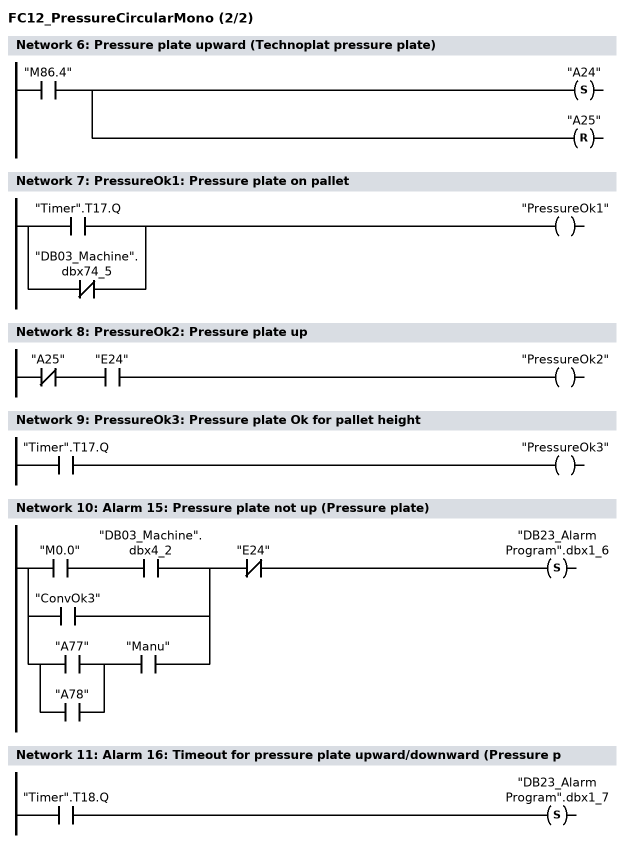
   RUNG wire#powerrail
      Contact( "M86.4" )
      wire#w1
      S_Coil( "A24" )
   END_RUNG
   RUNG wire#w1
      R_Coil( "A25" )
   END_RUNG
   // the same network as SCL:
   IF "M86.4" THEN
       "A24" := TRUE;
       "A25" := FALSE;
   END_IF;
END_REGION

REGION Network 7: PressureOk1: Pressure plate on pallet
   RUNG wire#powerrail
      Contact( "Timer".T17.Q )
      wire#w1
      Coil( "PressureOk1" )
   END_RUNG
   RUNG wire#powerrail
      I_Contact( "DB03_Machine".dbx74_5 )
   END_RUNG wire#w1
   // the same network as SCL:
   "PressureOk1" := "Timer".T17.Q OR NOT "DB03_Machine".dbx74_5;
END_REGION

REGION Network 8: PressureOk2: Pressure plate up
   RUNG wire#powerrail
      I_Contact( "A25" )
      Contact( "E24" )
      Coil( "PressureOk2" )
   END_RUNG
   // the same network as SCL:
   "PressureOk2" := NOT "A25" AND "E24";
END_REGION

REGION Network 9: PressureOk3: Pressure plate Ok for pallet height
   RUNG wire#powerrail
      Contact( "Timer".T17.Q )
      Coil( "PressureOk3" )
   END_RUNG
   // the same network as SCL:
   "PressureOk3" := "Timer".T17.Q;
END_REGION

REGION Network 10: Alarm 15: Pressure plate not up (Pressure plate)
   RUNG wire#powerrail
      Contact( "M0.0" )
      Contact( "DB03_Machine".dbx4_2 )
      wire#w1
      I_Contact( "E24" )
      S_Coil( "DB23_AlarmProgram".dbx1_6 )
   END_RUNG
   RUNG wire#powerrail
      Contact( "ConvOk3" )
   END_RUNG wire#w1
   RUNG wire#powerrail
      Contact( "A77" )
      wire#w2
      Contact( "Manu" )
   END_RUNG wire#w1
   RUNG wire#powerrail
      Contact( "A78" )
   END_RUNG wire#w2
   // the same network as SCL:
   IF (("M0.0" AND "DB03_Machine".dbx4_2) OR "ConvOk3" OR (("A77" OR "A78") AND "Manu")) AND NOT "E24" THEN
       "DB23_AlarmProgram".dbx1_6 := TRUE;
   END_IF;
END_REGION

REGION Network 11: Alarm 16: Timeout for pressure plate upward/downward (Pressure p
   RUNG wire#powerrail
      Contact( "Timer".T18.Q )
      S_Coil( "DB23_AlarmProgram".dbx1_7 )
   END_RUNG
   // the same network as SCL:
   IF "Timer".T18.Q THEN "DB23_AlarmProgram".dbx1_7 := TRUE; END_IF;
END_REGION
END_FUNCTION

FUNCTION "FC26_Pos1SensorDec" : Void   // FC26, LAD
{ S7_Optimized_Access := 'FALSE' }
VERSION : 0.1
// stored: AutoNumber false, IsIECCheckEnabled false, SetENOAutomatically false, UDAEnableTagReadback false
BEGIN

REGION Network 1: Delay on pallet positioning
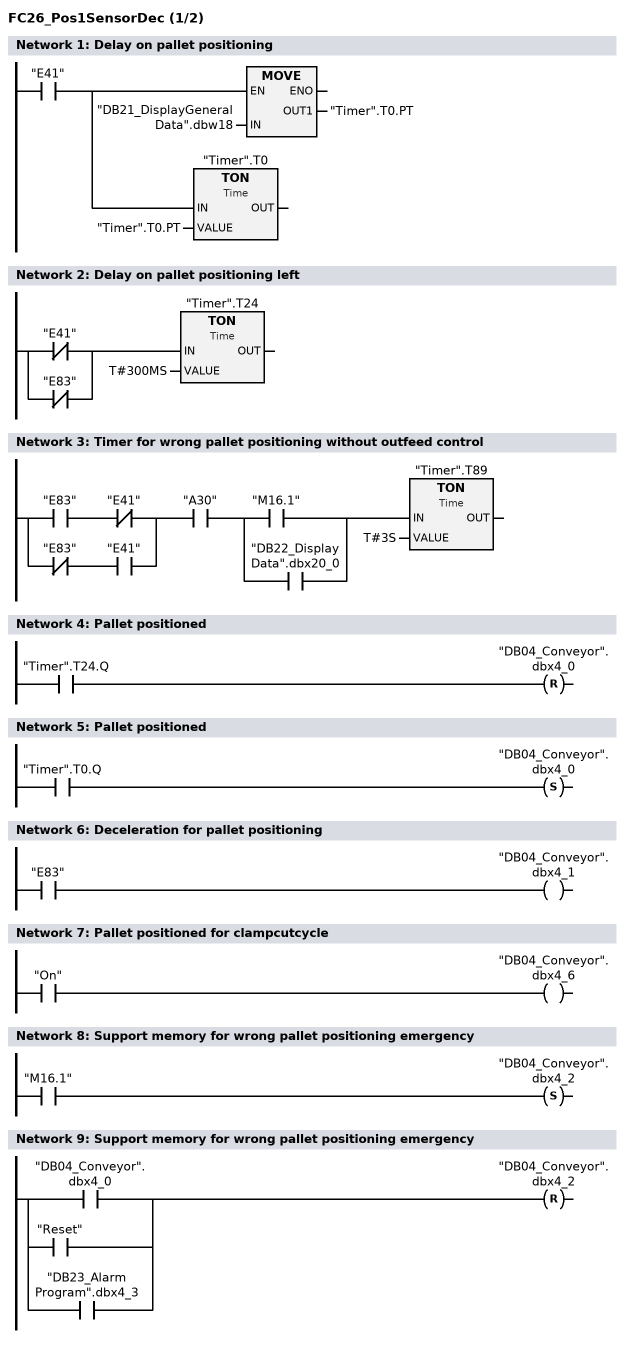
   IF "E41" THEN "Timer".T0.PT := "DB21_DisplayGeneralData".dbw18; END_IF;
   "Timer".T0.TON(IN := "E41", PT := "Timer".T0.PT);   // TON coil
END_REGION

REGION Network 2: Delay on pallet positioning left
   "Timer".T24.TON(IN := NOT "E41" OR NOT "E83", PT := T#300MS);   // TON coil
END_REGION

REGION Network 3: Timer for wrong pallet positioning without outfeed control
   "Timer".T89.TON(IN := (("E83" AND NOT "E41") OR (NOT "E83" AND "E41")) AND "A30" AND ("M16.1" OR "DB22_DisplayData".dbx20_0), PT := T#3S);   // TON coil
END_REGION

REGION Network 4: Pallet positioned
   RUNG wire#powerrail
      Contact( "Timer".T24.Q )
      R_Coil( "DB04_Conveyor".dbx4_0 )
   END_RUNG
   // the same network as SCL:
   IF "Timer".T24.Q THEN "DB04_Conveyor".dbx4_0 := FALSE; END_IF;
END_REGION

REGION Network 5: Pallet positioned
   RUNG wire#powerrail
      Contact( "Timer".T0.Q )
      S_Coil( "DB04_Conveyor".dbx4_0 )
   END_RUNG
   // the same network as SCL:
   IF "Timer".T0.Q THEN "DB04_Conveyor".dbx4_0 := TRUE; END_IF;
END_REGION

REGION Network 6: Deceleration for pallet positioning
   RUNG wire#powerrail
      Contact( "E83" )
      Coil( "DB04_Conveyor".dbx4_1 )
   END_RUNG
   // the same network as SCL:
   "DB04_Conveyor".dbx4_1 := "E83";
END_REGION

REGION Network 7: Pallet positioned for clampcutcycle
   RUNG wire#powerrail
      Contact( "On" )
      Coil( "DB04_Conveyor".dbx4_6 )
   END_RUNG
   // the same network as SCL:
   "DB04_Conveyor".dbx4_6 := "On";
END_REGION

REGION Network 8: Support memory for wrong pallet positioning emergency
   RUNG wire#powerrail
      Contact( "M16.1" )
      S_Coil( "DB04_Conveyor".dbx4_2 )
   END_RUNG
   // the same network as SCL:
   IF "M16.1" THEN "DB04_Conveyor".dbx4_2 := TRUE; END_IF;
END_REGION

REGION Network 9: Support memory for wrong pallet positioning emergency
   RUNG wire#powerrail
      Contact( "DB04_Conveyor".dbx4_0 )
      wire#w1
      R_Coil( "DB04_Conveyor".dbx4_2 )
   END_RUNG
   RUNG wire#powerrail
      Contact( "Reset" )
   END_RUNG wire#w1
   RUNG wire#powerrail
      Contact( "DB23_AlarmProgram".dbx4_3 )
   END_RUNG wire#w1
   // the same network as SCL:
   IF "DB04_Conveyor".dbx4_0 OR "Reset" OR "DB23_AlarmProgram".dbx4_3 THEN
       "DB04_Conveyor".dbx4_2 := FALSE;
   END_IF;
END_REGION

REGION Network 10: Alarm 33: Pallet positioning released during table rotation (Con
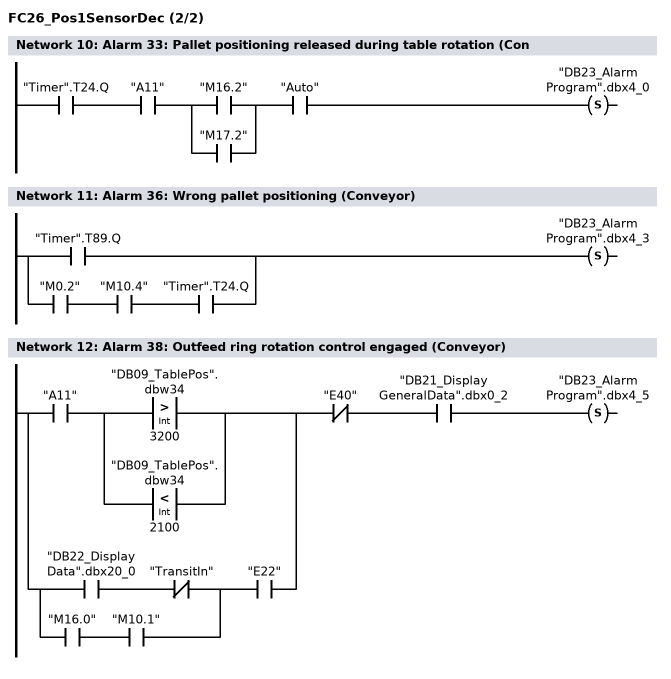
   RUNG wire#powerrail
      Contact( "Timer".T24.Q )
      Contact( "A11" )
      wire#w1
      Contact( "M16.2" )
      wire#w2
      Contact( "Auto" )
      S_Coil( "DB23_AlarmProgram".dbx4_0 )
   END_RUNG
   RUNG wire#w1
      Contact( "M17.2" )
   END_RUNG wire#w2
   // the same network as SCL:
   IF "Timer".T24.Q AND "A11" AND ("M16.2" OR "M17.2") AND "Auto" THEN
       "DB23_AlarmProgram".dbx4_0 := TRUE;
   END_IF;
END_REGION

REGION Network 11: Alarm 36: Wrong pallet positioning (Conveyor)
   RUNG wire#powerrail
      Contact( "Timer".T89.Q )
      wire#w1
      S_Coil( "DB23_AlarmProgram".dbx4_3 )
   END_RUNG
   RUNG wire#powerrail
      Contact( "M0.2" )
      Contact( "M10.4" )
      Contact( "Timer".T24.Q )
   END_RUNG wire#w1
   // the same network as SCL:
   IF "Timer".T89.Q OR ("M0.2" AND "M10.4" AND "Timer".T24.Q) THEN
       "DB23_AlarmProgram".dbx4_3 := TRUE;
   END_IF;
END_REGION

REGION Network 12: Alarm 38: Outfeed ring rotation control engaged (Conveyor)
   RUNG wire#powerrail
      Contact( "A11" )
      wire#w1
      { S7_Templates := "SrcType := Int" } GT_Contact(in1 := "DB09_TablePos".dbw34, in2 := 3200)
      wire#w2
      I_Contact( "E40" )
      Contact( "DB21_DisplayGeneralData".dbx0_2 )
      S_Coil( "DB23_AlarmProgram".dbx4_5 )
   END_RUNG
   RUNG wire#w1
      { S7_Templates := "SrcType := Int" } LT_Contact(in1 := "DB09_TablePos".dbw34, in2 := 2100)
   END_RUNG wire#w2
   RUNG wire#powerrail
      Contact( "DB22_DisplayData".dbx20_0 )
      I_Contact( "TransitIn" )
      wire#w3
      Contact( "E22" )
   END_RUNG wire#w2
   RUNG wire#powerrail
      Contact( "M16.0" )
      Contact( "M10.1" )
   END_RUNG wire#w3
   // the same network as SCL:
   IF (("A11" AND (("DB09_TablePos".dbw34 > 3200) OR ("DB09_TablePos".dbw34 < 2100))) OR ((("DB22_DisplayData".dbx20_0 AND NOT "TransitIn") OR ("M16.0" AND "M10.1")) AND "E22")) AND NOT "E40" AND "DB21_DisplayGeneralData".dbx0_2 THEN
       "DB23_AlarmProgram".dbx4_5 := TRUE;
   END_IF;
END_REGION
END_FUNCTION

FUNCTION "FC27_PosSelfcEncoder" : Void   // FC27, LAD
TITLE = Pallet positioning with selfcentering system and encoder
{ S7_Optimized_Access := 'FALSE' }
AUTHOR : Robopac
VERSION : 0.0
// stored: AutoNumber false, IsIECCheckEnabled false, SetENOAutomatically false, UDAEnableTagReadback false
   VAR_TEMP
      Ch7ValmmEnco1 : DInt;
      Ch7ValmmEnco2 : DInt;
      PalletLenghtdiv2 : Int;
      PosToReach : Int;
      PosToDecelation : Int;
      WTemp1 : Int;
      DWTemp1 : DInt;
      DWTemp2 : DInt;
   END_VAR
   VAR_TEMP   // added for the SCL form of the ladder/FBD networks
      _w1 : Bool;
      _w2 : Bool;
   END_VAR
BEGIN

REGION Network 1: Delay on pallet positioning left
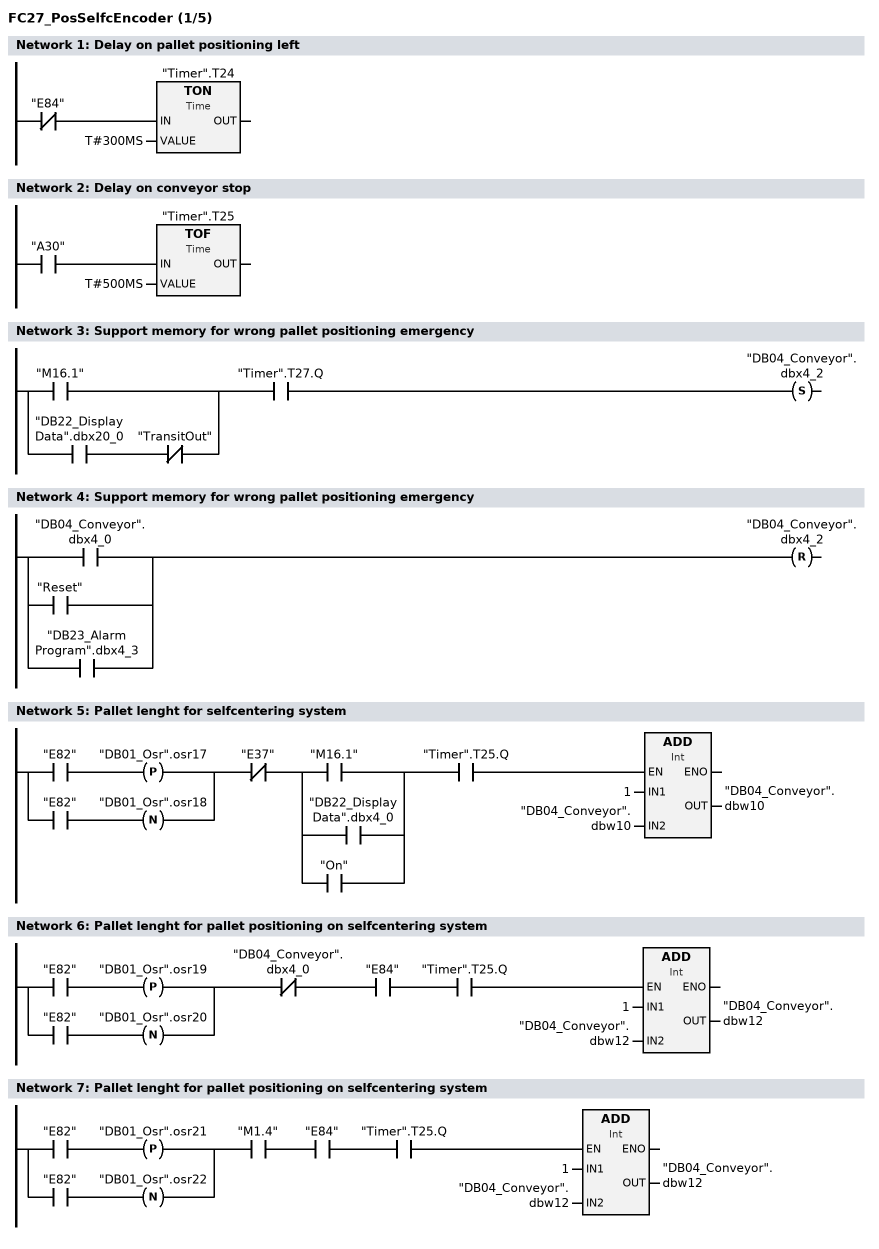
   "Timer".T24.TON(IN := NOT "E84", PT := T#300MS);   // TON coil
END_REGION

REGION Network 2: Delay on conveyor stop
   "Timer".T25.TOF(IN := "A30", PT := T#500MS);   // TOF coil
END_REGION

REGION Network 3: Support memory for wrong pallet positioning emergency
   RUNG wire#powerrail
      Contact( "M16.1" )
      wire#w1
      Contact( "Timer".T27.Q )
      S_Coil( "DB04_Conveyor".dbx4_2 )
   END_RUNG
   RUNG wire#powerrail
      Contact( "DB22_DisplayData".dbx20_0 )
      I_Contact( "TransitOut" )
   END_RUNG wire#w1
   // the same network as SCL:
   IF ("M16.1" OR ("DB22_DisplayData".dbx20_0 AND NOT "TransitOut")) AND "Timer".T27.Q THEN
       "DB04_Conveyor".dbx4_2 := TRUE;
   END_IF;
END_REGION

REGION Network 4: Support memory for wrong pallet positioning emergency
   RUNG wire#powerrail
      Contact( "DB04_Conveyor".dbx4_0 )
      wire#w1
      R_Coil( "DB04_Conveyor".dbx4_2 )
   END_RUNG
   RUNG wire#powerrail
      Contact( "Reset" )
   END_RUNG wire#w1
   RUNG wire#powerrail
      Contact( "DB23_AlarmProgram".dbx4_3 )
   END_RUNG wire#w1
   // the same network as SCL:
   IF "DB04_Conveyor".dbx4_0 OR "Reset" OR "DB23_AlarmProgram".dbx4_3 THEN
       "DB04_Conveyor".dbx4_2 := FALSE;
   END_IF;
END_REGION

REGION Network 5: Pallet lenght for selfcentering system
   RUNG wire#powerrail
      Contact( "E82" )
      P_Trig( "DB01_Osr".osr17 )
      wire#w1
      I_Contact( "E37" )
      wire#w2
      Contact( "M16.1" )
      wire#w3
      Contact( "Timer".T25.Q )
      { S7_Templates := "SrcType := Int"; S7_GenerateENO := "TRUE" } Add(in1 := 1, in2 := "DB04_Conveyor".dbw10, out => "DB04_Conveyor".dbw10)
   END_RUNG
   RUNG wire#powerrail
      Contact( "E82" )
      N_Trig( "DB01_Osr".osr18 )
   END_RUNG wire#w1
   RUNG wire#w2
      Contact( "DB22_DisplayData".dbx4_0 )
   END_RUNG wire#w3
   RUNG wire#w2
      Contact( "On" )
   END_RUNG wire#w3
   // the same network as SCL:
   #_w1 := "E82" AND NOT "DB01_Osr".osr17;   // rising edge
   "DB01_Osr".osr17 := "E82";
   #_w2 := NOT "E82" AND "DB01_Osr".osr18;   // falling edge
   "DB01_Osr".osr18 := "E82";
   IF (#_w1 OR #_w2) AND NOT "E37" AND ("M16.1" OR "DB22_DisplayData".dbx4_0 OR "On") AND "Timer".T25.Q THEN
       "DB04_Conveyor".dbw10 := 1 + "DB04_Conveyor".dbw10;
   END_IF;
END_REGION

REGION Network 6: Pallet lenght for pallet positioning on selfcentering system
   RUNG wire#powerrail
      Contact( "E82" )
      P_Trig( "DB01_Osr".osr19 )
      wire#w1
      I_Contact( "DB04_Conveyor".dbx4_0 )
      Contact( "E84" )
      Contact( "Timer".T25.Q )
      { S7_Templates := "SrcType := Int"; S7_GenerateENO := "TRUE" } Add(in1 := 1, in2 := "DB04_Conveyor".dbw12, out => "DB04_Conveyor".dbw12)
   END_RUNG
   RUNG wire#powerrail
      Contact( "E82" )
      N_Trig( "DB01_Osr".osr20 )
   END_RUNG wire#w1
   // the same network as SCL:
   #_w1 := "E82" AND NOT "DB01_Osr".osr19;   // rising edge
   "DB01_Osr".osr19 := "E82";
   #_w2 := NOT "E82" AND "DB01_Osr".osr20;   // falling edge
   "DB01_Osr".osr20 := "E82";
   IF (#_w1 OR #_w2) AND NOT "DB04_Conveyor".dbx4_0 AND "E84" AND "Timer".T25.Q THEN
       "DB04_Conveyor".dbw12 := 1 + "DB04_Conveyor".dbw12;
   END_IF;
END_REGION

REGION Network 7: Pallet lenght for pallet positioning on selfcentering system
   RUNG wire#powerrail
      Contact( "E82" )
      P_Trig( "DB01_Osr".osr21 )
      wire#w1
      Contact( "M1.4" )
      Contact( "E84" )
      Contact( "Timer".T25.Q )
      { S7_Templates := "SrcType := Int"; S7_GenerateENO := "TRUE" } Add(in1 := 1, in2 := "DB04_Conveyor".dbw12, out => "DB04_Conveyor".dbw12)
   END_RUNG
   RUNG wire#powerrail
      Contact( "E82" )
      N_Trig( "DB01_Osr".osr22 )
   END_RUNG wire#w1
   // the same network as SCL:
   #_w1 := "E82" AND NOT "DB01_Osr".osr21;   // rising edge
   "DB01_Osr".osr21 := "E82";
   #_w2 := NOT "E82" AND "DB01_Osr".osr22;   // falling edge
   "DB01_Osr".osr22 := "E82";
   IF (#_w1 OR #_w2) AND "M1.4" AND "E84" AND "Timer".T25.Q THEN
       "DB04_Conveyor".dbw12 := 1 + "DB04_Conveyor".dbw12;
   END_IF;
END_REGION

REGION Network 8: Reset pallet lenght
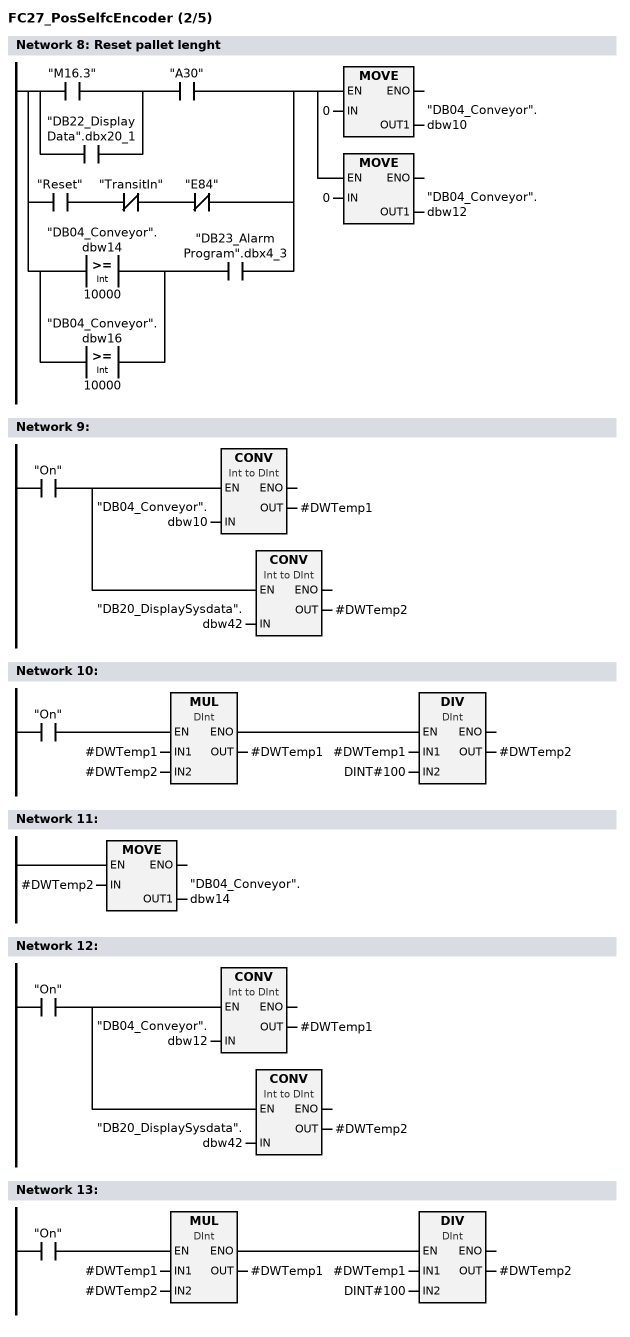
   RUNG wire#powerrail
      Contact( "M16.3" )
      wire#w1
      Contact( "A30" )
      wire#w2
      { S7_GenerateENO := "TRUE" } Move(in := 0, out1 => "DB04_Conveyor".dbw10)
   END_RUNG
   RUNG wire#powerrail
      Contact( "DB22_DisplayData".dbx20_1 )
   END_RUNG wire#w1
   RUNG wire#powerrail
      Contact( "Reset" )
      I_Contact( "TransitIn" )
      I_Contact( "E84" )
   END_RUNG wire#w2
   RUNG wire#powerrail
      { S7_Templates := "SrcType := Int" } GE_Contact(in1 := "DB04_Conveyor".dbw14, in2 := 10000)
      wire#w3
      Contact( "DB23_AlarmProgram".dbx4_3 )
   END_RUNG wire#w2
   RUNG wire#powerrail
      { S7_Templates := "SrcType := Int" } GE_Contact(in1 := "DB04_Conveyor".dbw16, in2 := 10000)
   END_RUNG wire#w3
   RUNG wire#w2
      { S7_GenerateENO := "TRUE" } Move(in := 0, out1 => "DB04_Conveyor".dbw12)
   END_RUNG
   // the same network as SCL:
   IF (("M16.3" OR "DB22_DisplayData".dbx20_1) AND "A30") OR ("Reset" AND NOT "TransitIn" AND NOT "E84") OR ((("DB04_Conveyor".dbw14 >= 10000) OR ("DB04_Conveyor".dbw16 >= 10000)) AND "DB23_AlarmProgram".dbx4_3) THEN
       "DB04_Conveyor".dbw10 := 0;
       "DB04_Conveyor".dbw12 := 0;
   END_IF;
END_REGION

REGION Network 9
   RUNG wire#powerrail
      Contact( "On" )
      wire#w1
      { S7_Templates := "[SrcType := Int, DestType := DInt]"; S7_GenerateENO := "TRUE" } Convert(in := "DB04_Conveyor".dbw10, out => #DWTemp1)
   END_RUNG
   RUNG wire#w1
      { S7_Templates := "[SrcType := Int, DestType := DInt]"; S7_GenerateENO := "TRUE" } Convert(in := "DB20_DisplaySysdata".dbw42, out => #DWTemp2)
   END_RUNG
   // the same network as SCL:
   IF "On" THEN
       #DWTemp1 := INT_TO_DINT("DB04_Conveyor".dbw10);
       #DWTemp2 := INT_TO_DINT("DB20_DisplaySysdata".dbw42);
   END_IF;
END_REGION

REGION Network 10
   RUNG wire#powerrail
      Contact( "On" )
      { S7_Templates := "SrcType := DInt"; S7_GenerateENO := "TRUE" } Mul(in1 := #DWTemp1, in2 := #DWTemp2, out => #DWTemp1)
      { S7_Templates := "SrcType := DInt"; S7_GenerateENO := "TRUE" } Div(in1 := #DWTemp1, in2 := DINT#100, out => #DWTemp2)
   END_RUNG
   // the same network as SCL:
   // ENO of a box is taken as its EN; it also drops when the box reports an error
   IF "On" THEN
       #DWTemp1 := #DWTemp1 * #DWTemp2;
       #DWTemp2 := #DWTemp1 / DINT#100;
   END_IF;
END_REGION

REGION Network 11
   RUNG wire#powerrail
      { S7_GenerateENO := "TRUE" } Move(in := #DWTemp2, out1 => "DB04_Conveyor".dbw14)
   END_RUNG
   // the same network as SCL:
   "DB04_Conveyor".dbw14 := #DWTemp2;
END_REGION

REGION Network 12
   RUNG wire#powerrail
      Contact( "On" )
      wire#w1
      { S7_Templates := "[SrcType := Int, DestType := DInt]"; S7_GenerateENO := "TRUE" } Convert(in := "DB04_Conveyor".dbw12, out => #DWTemp1)
   END_RUNG
   RUNG wire#w1
      { S7_Templates := "[SrcType := Int, DestType := DInt]"; S7_GenerateENO := "TRUE" } Convert(in := "DB20_DisplaySysdata".dbw42, out => #DWTemp2)
   END_RUNG
   // the same network as SCL:
   IF "On" THEN
       #DWTemp1 := INT_TO_DINT("DB04_Conveyor".dbw12);
       #DWTemp2 := INT_TO_DINT("DB20_DisplaySysdata".dbw42);
   END_IF;
END_REGION

REGION Network 13
   RUNG wire#powerrail
      Contact( "On" )
      { S7_Templates := "SrcType := DInt"; S7_GenerateENO := "TRUE" } Mul(in1 := #DWTemp1, in2 := #DWTemp2, out => #DWTemp1)
      { S7_Templates := "SrcType := DInt"; S7_GenerateENO := "TRUE" } Div(in1 := #DWTemp1, in2 := DINT#100, out => #DWTemp2)
   END_RUNG
   // the same network as SCL:
   // ENO of a box is taken as its EN; it also drops when the box reports an error
   IF "On" THEN
       #DWTemp1 := #DWTemp1 * #DWTemp2;
       #DWTemp2 := #DWTemp1 / DINT#100;
   END_IF;
END_REGION

REGION Network 14
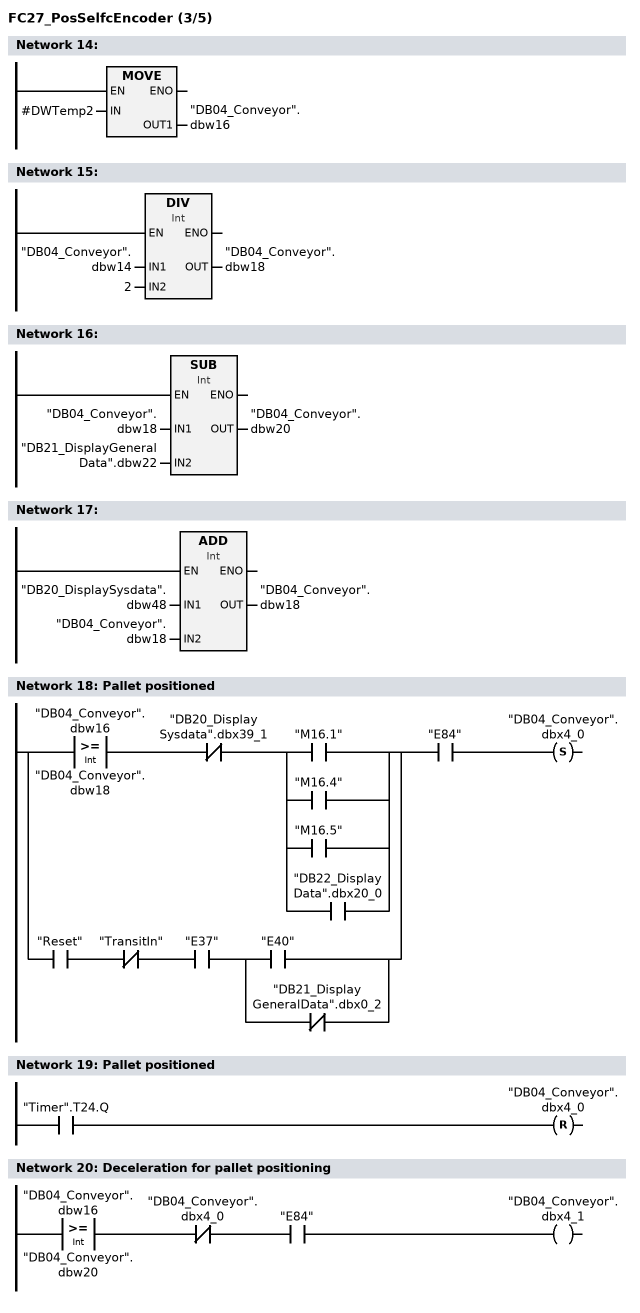
   RUNG wire#powerrail
      { S7_GenerateENO := "TRUE" } Move(in := #DWTemp2, out1 => "DB04_Conveyor".dbw16)
   END_RUNG
   // the same network as SCL:
   "DB04_Conveyor".dbw16 := #DWTemp2;
END_REGION

REGION Network 15
   RUNG wire#powerrail
      { S7_Templates := "SrcType := Int"; S7_GenerateENO := "TRUE" } Div(in1 := "DB04_Conveyor".dbw14, in2 := 2, out => "DB04_Conveyor".dbw18)
   END_RUNG
   // the same network as SCL:
   "DB04_Conveyor".dbw18 := "DB04_Conveyor".dbw14 / 2;
END_REGION

REGION Network 16
   RUNG wire#powerrail
      { S7_Templates := "SrcType := Int"; S7_GenerateENO := "TRUE" } Sub(in1 := "DB04_Conveyor".dbw18, in2 := "DB21_DisplayGeneralData".dbw22, out => "DB04_Conveyor".dbw20)
   END_RUNG
   // the same network as SCL:
   "DB04_Conveyor".dbw20 := "DB04_Conveyor".dbw18 - "DB21_DisplayGeneralData".dbw22;
END_REGION

REGION Network 17
   RUNG wire#powerrail
      { S7_Templates := "SrcType := Int"; S7_GenerateENO := "TRUE" } Add(in1 := "DB20_DisplaySysdata".dbw48, in2 := "DB04_Conveyor".dbw18, out => "DB04_Conveyor".dbw18)
   END_RUNG
   // the same network as SCL:
   "DB04_Conveyor".dbw18 := "DB20_DisplaySysdata".dbw48 + "DB04_Conveyor".dbw18;
END_REGION

REGION Network 18: Pallet positioned
   RUNG wire#powerrail
      { S7_Templates := "SrcType := Int" } GE_Contact(in1 := "DB04_Conveyor".dbw16, in2 := "DB04_Conveyor".dbw18)
      I_Contact( "DB20_DisplaySysdata".dbx39_1 )
      wire#w1
      Contact( "M16.1" )
      wire#w2
      Contact( "E84" )
      S_Coil( "DB04_Conveyor".dbx4_0 )
   END_RUNG
   RUNG wire#w1
      Contact( "M16.4" )
   END_RUNG wire#w2
   RUNG wire#w1
      Contact( "M16.5" )
   END_RUNG wire#w2
   RUNG wire#w1
      Contact( "DB22_DisplayData".dbx20_0 )
   END_RUNG wire#w2
   RUNG wire#powerrail
      Contact( "Reset" )
      I_Contact( "TransitIn" )
      Contact( "E37" )
      wire#w3
      Contact( "E40" )
   END_RUNG wire#w2
   RUNG wire#w3
      I_Contact( "DB21_DisplayGeneralData".dbx0_2 )
   END_RUNG wire#w2
   // the same network as SCL:
   IF ((("DB04_Conveyor".dbw16 >= "DB04_Conveyor".dbw18) AND NOT "DB20_DisplaySysdata".dbx39_1 AND ("M16.1" OR "M16.4" OR "M16.5" OR "DB22_DisplayData".dbx20_0)) OR ("Reset" AND NOT "TransitIn" AND "E37" AND ("E40" OR NOT "DB21_DisplayGeneralData".dbx0_2))) AND "E84" THEN
       "DB04_Conveyor".dbx4_0 := TRUE;
   END_IF;
END_REGION

REGION Network 19: Pallet positioned
   RUNG wire#powerrail
      Contact( "Timer".T24.Q )
      R_Coil( "DB04_Conveyor".dbx4_0 )
   END_RUNG
   // the same network as SCL:
   IF "Timer".T24.Q THEN "DB04_Conveyor".dbx4_0 := FALSE; END_IF;
END_REGION

REGION Network 20: Deceleration for pallet positioning
   RUNG wire#powerrail
      { S7_Templates := "SrcType := Int" } GE_Contact(in1 := "DB04_Conveyor".dbw16, in2 := "DB04_Conveyor".dbw20)
      I_Contact( "DB04_Conveyor".dbx4_0 )
      Contact( "E84" )
      Coil( "DB04_Conveyor".dbx4_1 )
   END_RUNG
   // the same network as SCL:
   "DB04_Conveyor".dbx4_1 := ("DB04_Conveyor".dbw16 >= "DB04_Conveyor".dbw20) AND NOT "DB04_Conveyor".dbx4_0 AND "E84";
END_REGION

REGION Network 21: Short pallet positioned
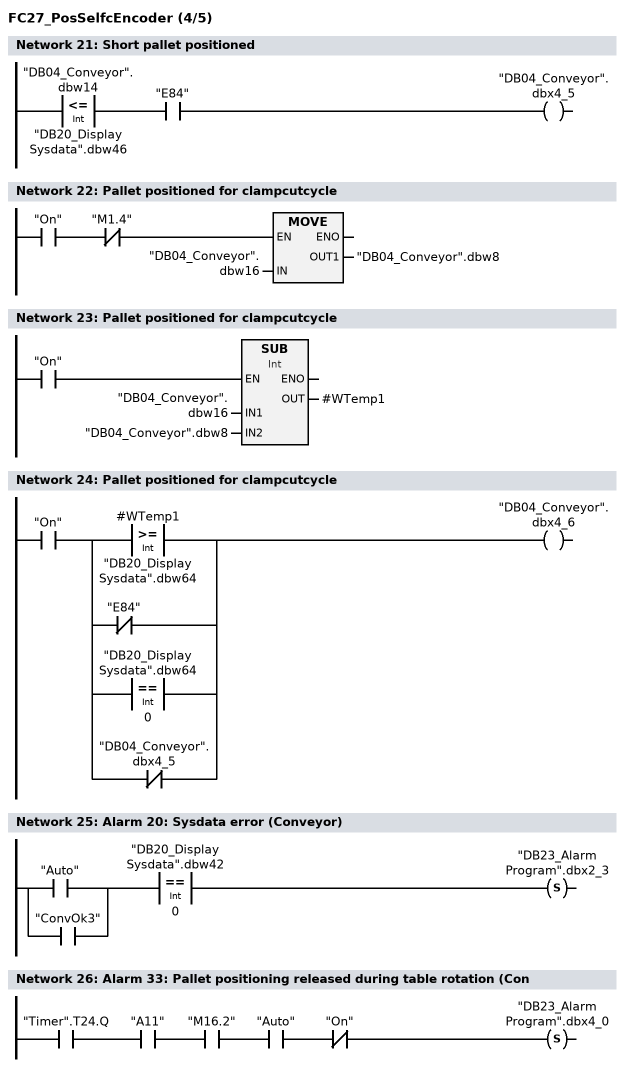
   RUNG wire#powerrail
      { S7_Templates := "SrcType := Int" } LE_Contact(in1 := "DB04_Conveyor".dbw14, in2 := "DB20_DisplaySysdata".dbw46)
      Contact( "E84" )
      Coil( "DB04_Conveyor".dbx4_5 )
   END_RUNG
   // the same network as SCL:
   "DB04_Conveyor".dbx4_5 := ("DB04_Conveyor".dbw14 <= "DB20_DisplaySysdata".dbw46) AND "E84";
END_REGION

REGION Network 22: Pallet positioned for clampcutcycle
   RUNG wire#powerrail
      Contact( "On" )
      I_Contact( "M1.4" )
      { S7_GenerateENO := "TRUE" } Move(in := "DB04_Conveyor".dbw16, out1 => "DB04_Conveyor".dbw8)
   END_RUNG
   // the same network as SCL:
   IF "On" AND NOT "M1.4" THEN "DB04_Conveyor".dbw8 := "DB04_Conveyor".dbw16; END_IF;
END_REGION

REGION Network 23: Pallet positioned for clampcutcycle
   RUNG wire#powerrail
      Contact( "On" )
      { S7_Templates := "SrcType := Int"; S7_GenerateENO := "TRUE" } Sub(in1 := "DB04_Conveyor".dbw16, in2 := "DB04_Conveyor".dbw8, out => #WTemp1)
   END_RUNG
   // the same network as SCL:
   IF "On" THEN #WTemp1 := "DB04_Conveyor".dbw16 - "DB04_Conveyor".dbw8; END_IF;
END_REGION

REGION Network 24: Pallet positioned for clampcutcycle
   RUNG wire#powerrail
      Contact( "On" )
      wire#w1
      { S7_Templates := "SrcType := Int" } GE_Contact(in1 := #WTemp1, in2 := "DB20_DisplaySysdata".dbw64)
      wire#w2
      Coil( "DB04_Conveyor".dbx4_6 )
   END_RUNG
   RUNG wire#w1
      I_Contact( "E84" )
   END_RUNG wire#w2
   RUNG wire#w1
      { S7_Templates := "SrcType := Int" } EQ_Contact(in1 := "DB20_DisplaySysdata".dbw64, in2 := 0)
   END_RUNG wire#w2
   RUNG wire#w1
      I_Contact( "DB04_Conveyor".dbx4_5 )
   END_RUNG wire#w2
   // the same network as SCL:
   "DB04_Conveyor".dbx4_6 := "On" AND ((#WTemp1 >= "DB20_DisplaySysdata".dbw64) OR NOT "E84" OR ("DB20_DisplaySysdata".dbw64 = 0) OR NOT "DB04_Conveyor".dbx4_5);
END_REGION

REGION Network 25: Alarm 20: Sysdata error (Conveyor)
   RUNG wire#powerrail
      Contact( "Auto" )
      wire#w1
      { S7_Templates := "SrcType := Int" } EQ_Contact(in1 := "DB20_DisplaySysdata".dbw42, in2 := 0)
      S_Coil( "DB23_AlarmProgram".dbx2_3 )
   END_RUNG
   RUNG wire#powerrail
      Contact( "ConvOk3" )
   END_RUNG wire#w1
   // the same network as SCL:
   IF ("Auto" OR "ConvOk3") AND ("DB20_DisplaySysdata".dbw42 = 0) THEN
       "DB23_AlarmProgram".dbx2_3 := TRUE;
   END_IF;
END_REGION

REGION Network 26: Alarm 33: Pallet positioning released during table rotation (Con
   RUNG wire#powerrail
      Contact( "Timer".T24.Q )
      Contact( "A11" )
      Contact( "M16.2" )
      Contact( "Auto" )
      I_Contact( "On" )
      S_Coil( "DB23_AlarmProgram".dbx4_0 )
   END_RUNG
   // the same network as SCL:
   IF "Timer".T24.Q AND "A11" AND "M16.2" AND "Auto" AND NOT "On" THEN
       "DB23_AlarmProgram".dbx4_0 := TRUE;
   END_IF;
END_REGION

REGION Network 27: Alarm 36: Wrong pallet positioning (Conveyor)
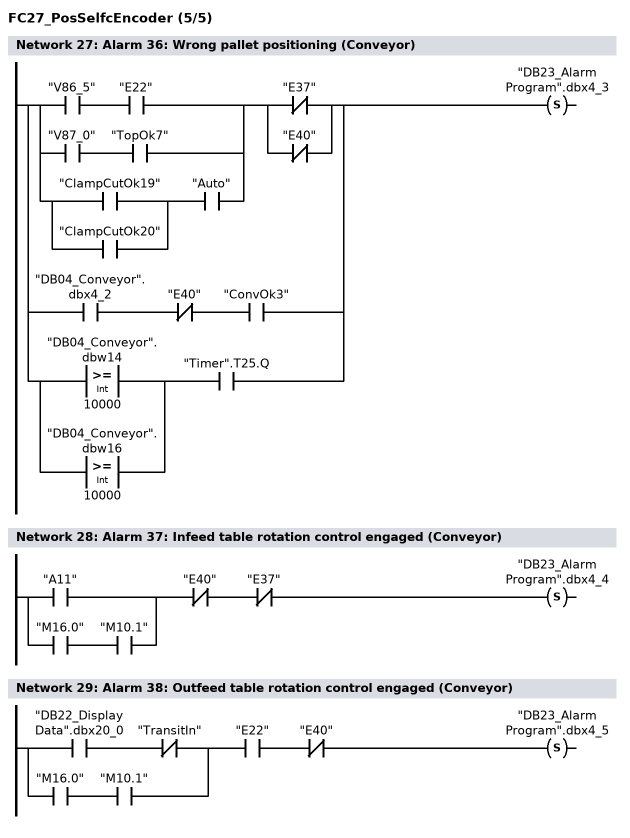
   RUNG wire#powerrail
      Contact( "V86_5" )
      Contact( "E22" )
      wire#w1
      I_Contact( "E37" )
      wire#w3
      S_Coil( "DB23_AlarmProgram".dbx4_3 )
   END_RUNG
   RUNG wire#powerrail
      Contact( "V87_0" )
      Contact( "TopOk7" )
   END_RUNG wire#w1
   RUNG wire#powerrail
      Contact( "ClampCutOk19" )
      wire#w2
      Contact( "Auto" )
   END_RUNG wire#w1
   RUNG wire#powerrail
      Contact( "ClampCutOk20" )
   END_RUNG wire#w2
   RUNG wire#w1
      I_Contact( "E40" )
   END_RUNG wire#w3
   RUNG wire#powerrail
      Contact( "DB04_Conveyor".dbx4_2 )
      I_Contact( "E40" )
      Contact( "ConvOk3" )
   END_RUNG wire#w3
   RUNG wire#powerrail
      { S7_Templates := "SrcType := Int" } GE_Contact(in1 := "DB04_Conveyor".dbw14, in2 := 10000)
      wire#w4
      Contact( "Timer".T25.Q )
   END_RUNG wire#w3
   RUNG wire#powerrail
      { S7_Templates := "SrcType := Int" } GE_Contact(in1 := "DB04_Conveyor".dbw16, in2 := 10000)
   END_RUNG wire#w4
   // the same network as SCL:
   IF ((("V86_5" AND "E22") OR ("V87_0" AND "TopOk7") OR (("ClampCutOk19" OR "ClampCutOk20") AND "Auto")) AND (NOT "E37" OR NOT "E40")) OR ("DB04_Conveyor".dbx4_2 AND NOT "E40" AND "ConvOk3") OR ((("DB04_Conveyor".dbw14 >= 10000) OR ("DB04_Conveyor".dbw16 >= 10000)) AND "Timer".T25.Q) THEN
       "DB23_AlarmProgram".dbx4_3 := TRUE;
   END_IF;
END_REGION

REGION Network 28: Alarm 37: Infeed table rotation control engaged (Conveyor)
   RUNG wire#powerrail
      Contact( "A11" )
      wire#w1
      I_Contact( "E40" )
      I_Contact( "E37" )
      S_Coil( "DB23_AlarmProgram".dbx4_4 )
   END_RUNG
   RUNG wire#powerrail
      Contact( "M16.0" )
      Contact( "M10.1" )
   END_RUNG wire#w1
   // the same network as SCL:
   IF ("A11" OR ("M16.0" AND "M10.1")) AND NOT "E40" AND NOT "E37" THEN
       "DB23_AlarmProgram".dbx4_4 := TRUE;
   END_IF;
END_REGION

REGION Network 29: Alarm 38: Outfeed table rotation control engaged (Conveyor)
   RUNG wire#powerrail
      Contact( "DB22_DisplayData".dbx20_0 )
      I_Contact( "TransitIn" )
      wire#w1
      Contact( "E22" )
      I_Contact( "E40" )
      S_Coil( "DB23_AlarmProgram".dbx4_5 )
   END_RUNG
   RUNG wire#powerrail
      Contact( "M16.0" )
      Contact( "M10.1" )
   END_RUNG wire#w1
   // the same network as SCL:
   IF (("DB22_DisplayData".dbx20_0 AND NOT "TransitIn") OR ("M16.0" AND "M10.1")) AND "E22" AND NOT "E40" THEN
       "DB23_AlarmProgram".dbx4_5 := TRUE;
   END_IF;
END_REGION
END_FUNCTION

FUNCTION "FC31_ConveyorInverter" : Void   // FC31, LAD
TITLE = Conveyor management with inverter
{ S7_Optimized_Access := 'FALSE' }
AUTHOR : Robopac
VERSION : 0.0
// stored: AutoNumber false, IsIECCheckEnabled false, SetENOAutomatically false, UDAEnableTagReadback false
   VAR_TEMP
      TimeUpwardTableCycle : Word;
      TimeUpwardTableCycleInt : Int;
      TempWord : Word;
   END_VAR
   VAR_TEMP   // added for the SCL form of the ladder/FBD networks
      _w1 : Bool;
   END_VAR
BEGIN

REGION Network 1: Timer SA type for conveyor motor
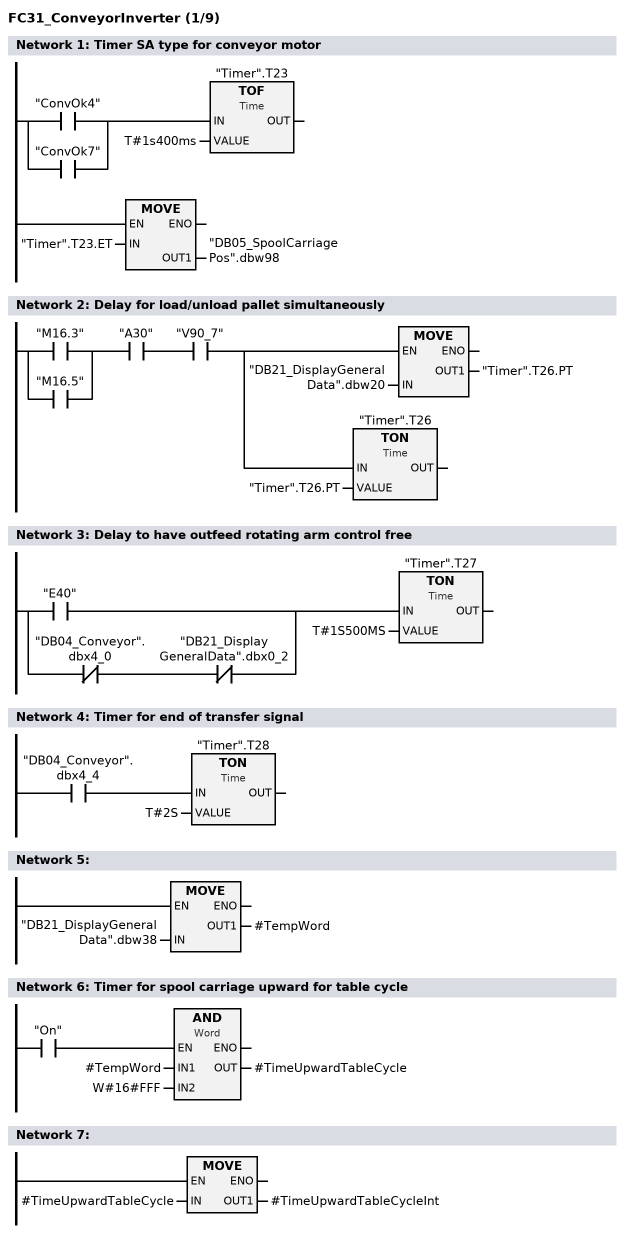
   "Timer".T23.TOF(IN := "ConvOk4" OR "ConvOk7", PT := T#1s400ms);   // TOF coil
   "DB05_SpoolCarriagePos".dbw98 := "Timer".T23.ET;
END_REGION

REGION Network 2: Delay for load/unload pallet simultaneously
   #_w1 := ("M16.3" OR "M16.5") AND "A30" AND "V90_7";
   IF #_w1 THEN "Timer".T26.PT := "DB21_DisplayGeneralData".dbw20; END_IF;
   "Timer".T26.TON(IN := #_w1, PT := "Timer".T26.PT);   // TON coil
END_REGION

REGION Network 3: Delay to have outfeed rotating arm control free
   "Timer".T27.TON(IN := "E40" OR (NOT "DB04_Conveyor".dbx4_0 AND NOT "DB21_DisplayGeneralData".dbx0_2), PT := T#1S500MS);   // TON coil
END_REGION

REGION Network 4: Timer for end of transfer signal
   "Timer".T28.TON(IN := "DB04_Conveyor".dbx4_4, PT := T#2S);   // TON coil
END_REGION

REGION Network 5
   RUNG wire#powerrail
      { S7_GenerateENO := "TRUE" } Move(in := "DB21_DisplayGeneralData".dbw38, out1 => #TempWord)
   END_RUNG
   // the same network as SCL:
   #TempWord := "DB21_DisplayGeneralData".dbw38;
END_REGION

REGION Network 6: Timer for spool carriage upward for table cycle
   RUNG wire#powerrail
      Contact( "On" )
      { S7_Templates := "SrcType := Word"; S7_GenerateENO := "TRUE" } And(in1 := #TempWord, in2 := W#16#FFF, out => #TimeUpwardTableCycle)
   END_RUNG
   // the same network as SCL:
   IF "On" THEN #TimeUpwardTableCycle := #TempWord AND W#16#FFF; END_IF;
END_REGION

REGION Network 7
   RUNG wire#powerrail
      { S7_GenerateENO := "TRUE" } Move(in := #TimeUpwardTableCycle, out1 => #TimeUpwardTableCycleInt)
   END_RUNG
   // the same network as SCL:
   #TimeUpwardTableCycleInt := #TimeUpwardTableCycle;
END_REGION

REGION Network 8: Timer for spool carriage upward for table cycle
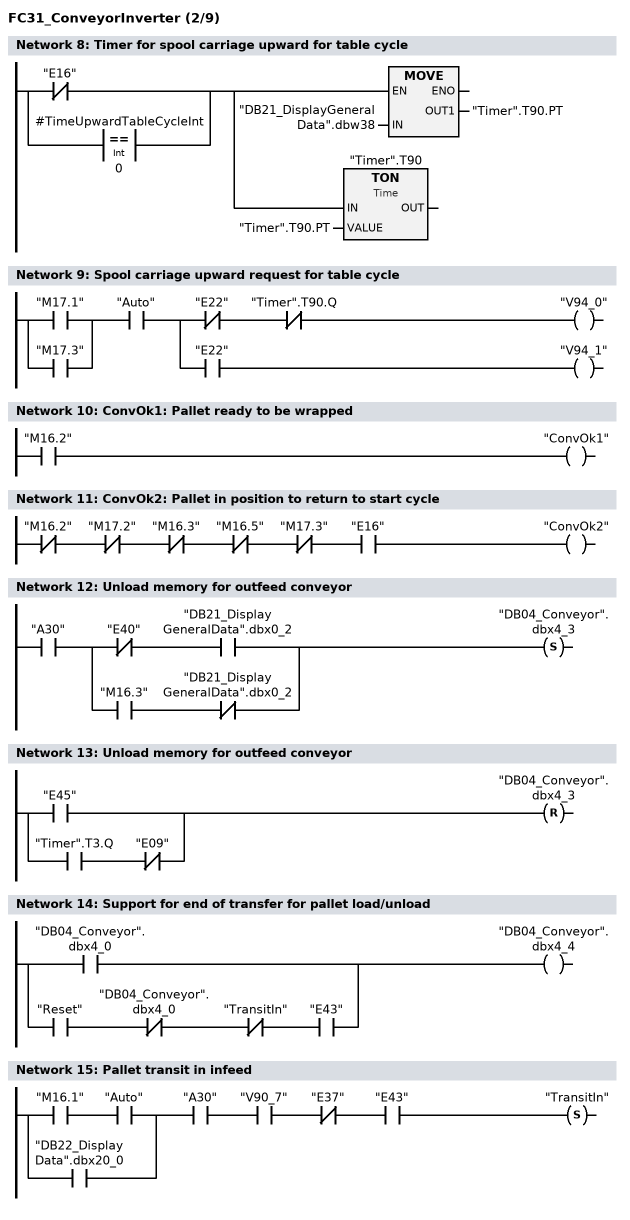
   #_w1 := NOT "E16" OR (#TimeUpwardTableCycleInt = 0);
   IF #_w1 THEN "Timer".T90.PT := "DB21_DisplayGeneralData".dbw38; END_IF;
   "Timer".T90.TON(IN := #_w1, PT := "Timer".T90.PT);   // TON coil
END_REGION

REGION Network 9: Spool carriage upward request for table cycle
   RUNG wire#powerrail
      Contact( "M17.1" )
      wire#w1
      Contact( "Auto" )
      wire#w2
      I_Contact( "E22" )
      I_Contact( "Timer".T90.Q )
      Coil( "V94_0" )
   END_RUNG
   RUNG wire#powerrail
      Contact( "M17.3" )
   END_RUNG wire#w1
   RUNG wire#w2
      Contact( "E22" )
      Coil( "V94_1" )
   END_RUNG
   // the same network as SCL:
   #_w1 := ("M17.1" OR "M17.3") AND "Auto";
   "V94_0" := #_w1 AND NOT "E22" AND NOT "Timer".T90.Q;
   "V94_1" := #_w1 AND "E22";
END_REGION

REGION Network 10: ConvOk1: Pallet ready to be wrapped
   RUNG wire#powerrail
      Contact( "M16.2" )
      Coil( "ConvOk1" )
   END_RUNG
   // the same network as SCL:
   "ConvOk1" := "M16.2";
END_REGION

REGION Network 11: ConvOk2: Pallet in position to return to start cycle
   RUNG wire#powerrail
      I_Contact( "M16.2" )
      I_Contact( "M17.2" )
      I_Contact( "M16.3" )
      I_Contact( "M16.5" )
      I_Contact( "M17.3" )
      Contact( "E16" )
      Coil( "ConvOk2" )
   END_RUNG
   // the same network as SCL:
   "ConvOk2" := NOT "M16.2" AND NOT "M17.2" AND NOT "M16.3" AND NOT "M16.5" AND NOT "M17.3" AND "E16";
END_REGION

REGION Network 12: Unload memory for outfeed conveyor
   RUNG wire#powerrail
      Contact( "A30" )
      wire#w1
      I_Contact( "E40" )
      Contact( "DB21_DisplayGeneralData".dbx0_2 )
      wire#w2
      S_Coil( "DB04_Conveyor".dbx4_3 )
   END_RUNG
   RUNG wire#w1
      Contact( "M16.3" )
      I_Contact( "DB21_DisplayGeneralData".dbx0_2 )
   END_RUNG wire#w2
   // the same network as SCL:
   IF "A30" AND ((NOT "E40" AND "DB21_DisplayGeneralData".dbx0_2) OR ("M16.3" AND NOT "DB21_DisplayGeneralData".dbx0_2)) THEN
       "DB04_Conveyor".dbx4_3 := TRUE;
   END_IF;
END_REGION

REGION Network 13: Unload memory for outfeed conveyor
   RUNG wire#powerrail
      Contact( "E45" )
      wire#w1
      R_Coil( "DB04_Conveyor".dbx4_3 )
   END_RUNG
   RUNG wire#powerrail
      Contact( "Timer".T3.Q )
      I_Contact( "E09" )
   END_RUNG wire#w1
   // the same network as SCL:
   IF "E45" OR ("Timer".T3.Q AND NOT "E09") THEN "DB04_Conveyor".dbx4_3 := FALSE; END_IF;
END_REGION

REGION Network 14: Support for end of transfer for pallet load/unload
   RUNG wire#powerrail
      Contact( "DB04_Conveyor".dbx4_0 )
      wire#w1
      Coil( "DB04_Conveyor".dbx4_4 )
   END_RUNG
   RUNG wire#powerrail
      Contact( "Reset" )
      I_Contact( "DB04_Conveyor".dbx4_0 )
      I_Contact( "TransitIn" )
      Contact( "E43" )
   END_RUNG wire#w1
   // the same network as SCL:
   "DB04_Conveyor".dbx4_4 := "DB04_Conveyor".dbx4_0 OR ("Reset" AND NOT "DB04_Conveyor".dbx4_0 AND NOT "TransitIn" AND "E43");
END_REGION

REGION Network 15: Pallet transit in infeed
   RUNG wire#powerrail
      Contact( "M16.1" )
      Contact( "Auto" )
      wire#w1
      Contact( "A30" )
      Contact( "V90_7" )
      I_Contact( "E37" )
      Contact( "E43" )
      S_Coil( "TransitIn" )
   END_RUNG
   RUNG wire#powerrail
      Contact( "DB22_DisplayData".dbx20_0 )
   END_RUNG wire#w1
   // the same network as SCL:
   IF (("M16.1" AND "Auto") OR "DB22_DisplayData".dbx20_0) AND "A30" AND "V90_7" AND NOT "E37" AND "E43" THEN
       "TransitIn" := TRUE;
   END_IF;
END_REGION

REGION Network 16: Pallet transit in infeed
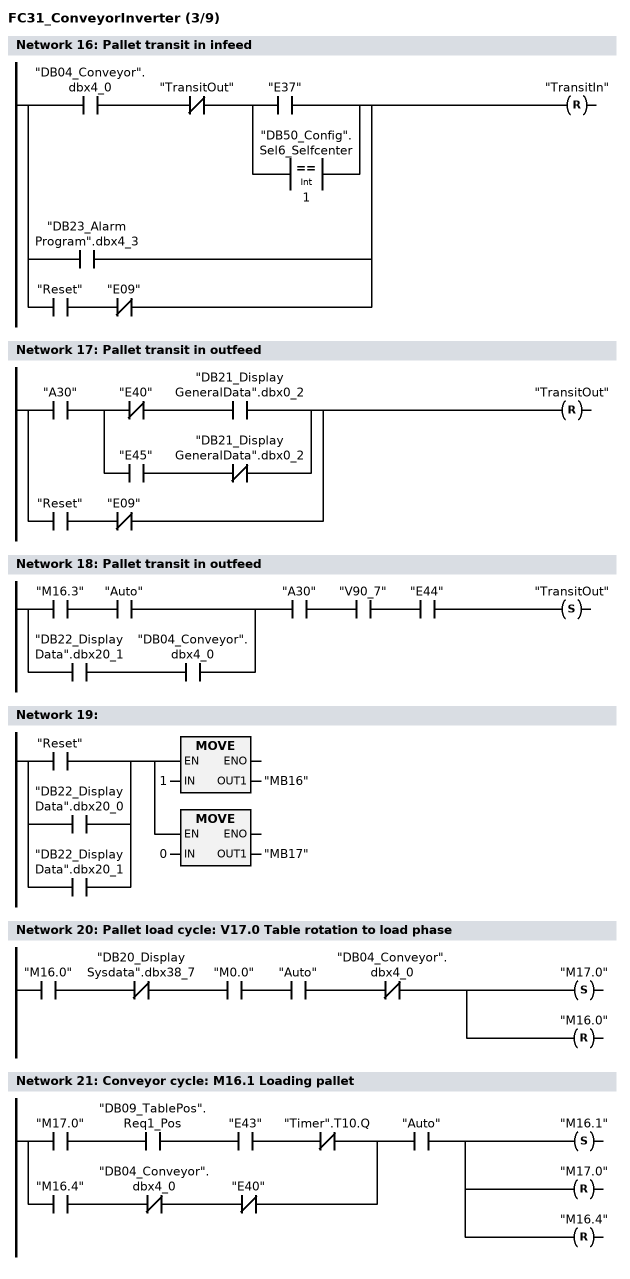
   IF ("DB04_Conveyor".dbx4_0 AND NOT "TransitOut" AND (("DB50_Config".Sel6_Selfcenter = 1) OR "E37")) OR "DB23_AlarmProgram".dbx4_3 OR ("Reset" AND NOT "E09") THEN
       "TransitIn" := FALSE;
   END_IF;
END_REGION

REGION Network 17: Pallet transit in outfeed
   RUNG wire#powerrail
      Contact( "A30" )
      wire#w1
      I_Contact( "E40" )
      Contact( "DB21_DisplayGeneralData".dbx0_2 )
      wire#w2
      R_Coil( "TransitOut" )
   END_RUNG
   RUNG wire#w1
      Contact( "E45" )
      I_Contact( "DB21_DisplayGeneralData".dbx0_2 )
   END_RUNG wire#w2
   RUNG wire#powerrail
      Contact( "Reset" )
      I_Contact( "E09" )
   END_RUNG wire#w2
   // the same network as SCL:
   IF ("A30" AND ((NOT "E40" AND "DB21_DisplayGeneralData".dbx0_2) OR ("E45" AND NOT "DB21_DisplayGeneralData".dbx0_2))) OR ("Reset" AND NOT "E09") THEN
       "TransitOut" := FALSE;
   END_IF;
END_REGION

REGION Network 18: Pallet transit in outfeed
   RUNG wire#powerrail
      Contact( "M16.3" )
      Contact( "Auto" )
      wire#w1
      Contact( "A30" )
      Contact( "V90_7" )
      Contact( "E44" )
      S_Coil( "TransitOut" )
   END_RUNG
   RUNG wire#powerrail
      Contact( "DB22_DisplayData".dbx20_1 )
      Contact( "DB04_Conveyor".dbx4_0 )
   END_RUNG wire#w1
   // the same network as SCL:
   IF (("M16.3" AND "Auto") OR ("DB22_DisplayData".dbx20_1 AND "DB04_Conveyor".dbx4_0)) AND "A30" AND "V90_7" AND "E44" THEN
       "TransitOut" := TRUE;
   END_IF;
END_REGION

REGION Network 19
   RUNG wire#powerrail
      Contact( "Reset" )
      wire#w1
      { S7_GenerateENO := "TRUE" } Move(in := 1, out1 => "MB16")
   END_RUNG
   RUNG wire#powerrail
      Contact( "DB22_DisplayData".dbx20_0 )
   END_RUNG wire#w1
   RUNG wire#powerrail
      Contact( "DB22_DisplayData".dbx20_1 )
   END_RUNG wire#w1
   RUNG wire#w1
      { S7_GenerateENO := "TRUE" } Move(in := 0, out1 => "MB17")
   END_RUNG
   // the same network as SCL:
   IF "Reset" OR "DB22_DisplayData".dbx20_0 OR "DB22_DisplayData".dbx20_1 THEN
       "MB16" := 1;
       "MB17" := 0;
   END_IF;
END_REGION

REGION Network 20: Pallet load cycle: V17.0 Table rotation to load phase
   RUNG wire#powerrail
      Contact( "M16.0" )
      I_Contact( "DB20_DisplaySysdata".dbx38_7 )
      Contact( "M0.0" )
      Contact( "Auto" )
      I_Contact( "DB04_Conveyor".dbx4_0 )
      wire#w1
      S_Coil( "M17.0" )
   END_RUNG
   RUNG wire#w1
      R_Coil( "M16.0" )
   END_RUNG
   // the same network as SCL:
   IF "M16.0" AND NOT "DB20_DisplaySysdata".dbx38_7 AND "M0.0" AND "Auto" AND NOT "DB04_Conveyor".dbx4_0 THEN
       "M17.0" := TRUE;
       "M16.0" := FALSE;
   END_IF;
END_REGION

REGION Network 21: Conveyor cycle: M16.1 Loading pallet
   RUNG wire#powerrail
      Contact( "M17.0" )
      Contact( "DB09_TablePos".Req1_Pos )
      Contact( "E43" )
      I_Contact( "Timer".T10.Q )
      wire#w1
      Contact( "Auto" )
      wire#w2
      S_Coil( "M16.1" )
   END_RUNG
   RUNG wire#powerrail
      Contact( "M16.4" )
      I_Contact( "DB04_Conveyor".dbx4_0 )
      I_Contact( "E40" )
   END_RUNG wire#w1
   RUNG wire#w2
      R_Coil( "M17.0" )
   END_RUNG
   RUNG wire#w2
      R_Coil( "M16.4" )
   END_RUNG
   // the same network as SCL:
   IF (("M17.0" AND "DB09_TablePos".Req1_Pos AND "E43" AND NOT "Timer".T10.Q) OR ("M16.4" AND NOT "DB04_Conveyor".dbx4_0 AND NOT "E40")) AND "Auto" THEN
       "M16.1" := TRUE;
   END_IF;
   #_w1 := (("M17.0" AND "DB09_TablePos".Req1_Pos AND "E43" AND NOT "Timer".T10.Q) OR ("M16.4" AND NOT "DB04_Conveyor".dbx4_0 AND NOT "E40")) AND "Auto";
   IF #_w1 THEN
       "M17.0" := FALSE;
       "M16.4" := FALSE;
   END_IF;
END_REGION

REGION Network 22: Pallet load cycle: V17.1 Table rotation to machine phase from lo
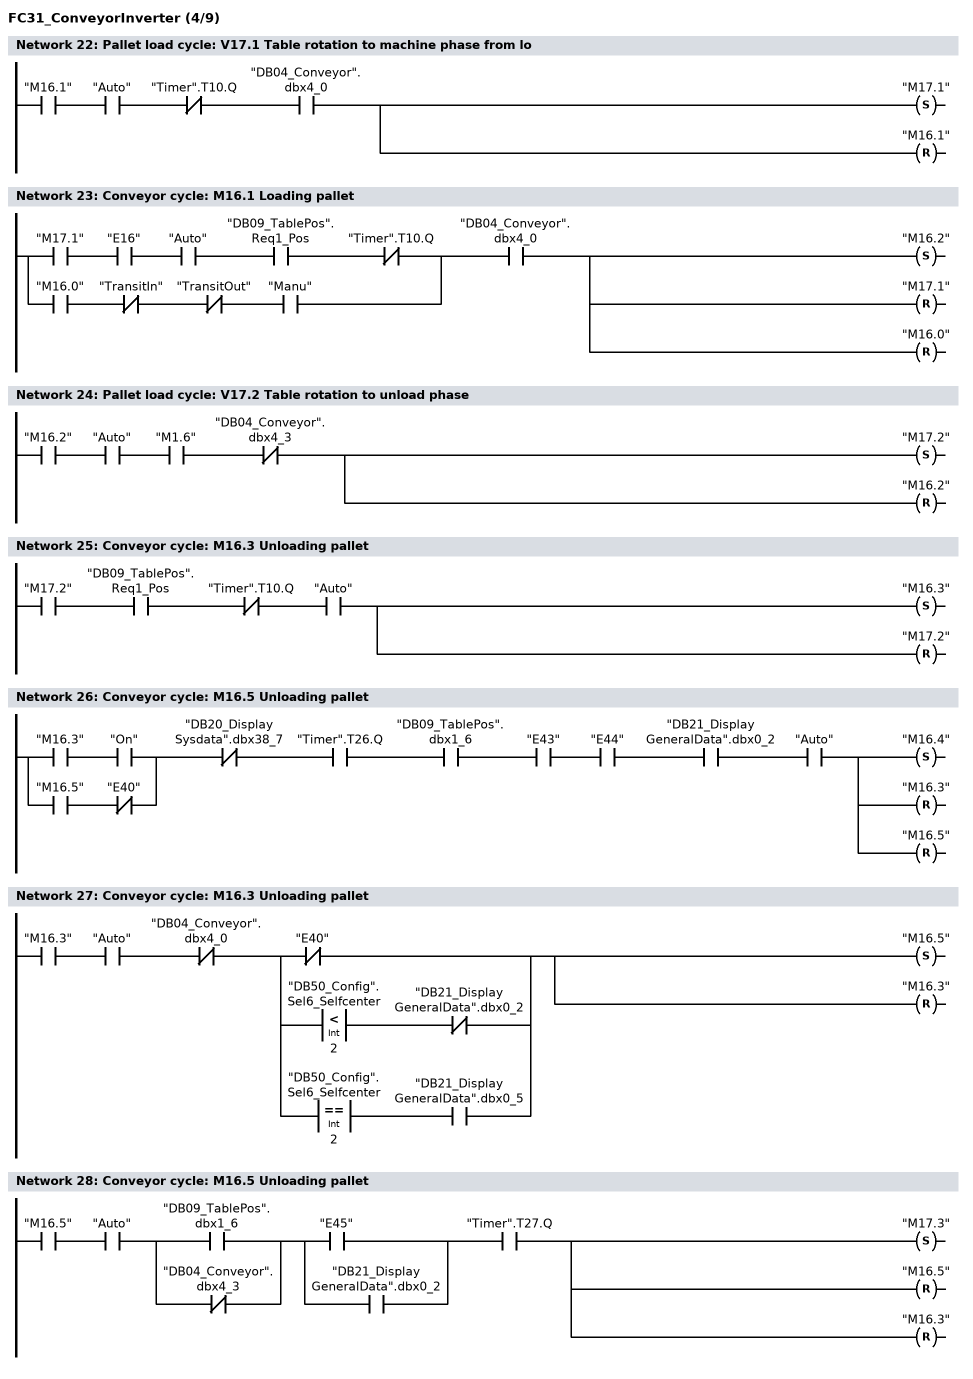
   RUNG wire#powerrail
      Contact( "M16.1" )
      Contact( "Auto" )
      I_Contact( "Timer".T10.Q )
      Contact( "DB04_Conveyor".dbx4_0 )
      wire#w1
      S_Coil( "M17.1" )
   END_RUNG
   RUNG wire#w1
      R_Coil( "M16.1" )
   END_RUNG
   // the same network as SCL:
   IF "M16.1" AND "Auto" AND NOT "Timer".T10.Q AND "DB04_Conveyor".dbx4_0 THEN
       "M17.1" := TRUE;
       "M16.1" := FALSE;
   END_IF;
END_REGION

REGION Network 23: Conveyor cycle: M16.1 Loading pallet
   RUNG wire#powerrail
      Contact( "M17.1" )
      Contact( "E16" )
      Contact( "Auto" )
      Contact( "DB09_TablePos".Req1_Pos )
      I_Contact( "Timer".T10.Q )
      wire#w1
      Contact( "DB04_Conveyor".dbx4_0 )
      wire#w2
      S_Coil( "M16.2" )
   END_RUNG
   RUNG wire#powerrail
      Contact( "M16.0" )
      I_Contact( "TransitIn" )
      I_Contact( "TransitOut" )
      Contact( "Manu" )
   END_RUNG wire#w1
   RUNG wire#w2
      R_Coil( "M17.1" )
   END_RUNG
   RUNG wire#w2
      R_Coil( "M16.0" )
   END_RUNG
   // the same network as SCL:
   IF (("M17.1" AND "E16" AND "Auto" AND "DB09_TablePos".Req1_Pos AND NOT "Timer".T10.Q) OR ("M16.0" AND NOT "TransitIn" AND NOT "TransitOut" AND "Manu")) AND "DB04_Conveyor".dbx4_0 THEN
       "M16.2" := TRUE;
   END_IF;
   #_w1 := (("M17.1" AND "E16" AND "Auto" AND "DB09_TablePos".Req1_Pos AND NOT "Timer".T10.Q) OR ("M16.0" AND NOT "TransitIn" AND NOT "TransitOut" AND "Manu")) AND "DB04_Conveyor".dbx4_0;
   IF #_w1 THEN
       "M17.1" := FALSE;
       "M16.0" := FALSE;
   END_IF;
END_REGION

REGION Network 24: Pallet load cycle: V17.2 Table rotation to unload phase
   RUNG wire#powerrail
      Contact( "M16.2" )
      Contact( "Auto" )
      Contact( "M1.6" )
      I_Contact( "DB04_Conveyor".dbx4_3 )
      wire#w1
      S_Coil( "M17.2" )
   END_RUNG
   RUNG wire#w1
      R_Coil( "M16.2" )
   END_RUNG
   // the same network as SCL:
   IF "M16.2" AND "Auto" AND "M1.6" AND NOT "DB04_Conveyor".dbx4_3 THEN
       "M17.2" := TRUE;
       "M16.2" := FALSE;
   END_IF;
END_REGION

REGION Network 25: Conveyor cycle: M16.3 Unloading pallet
   RUNG wire#powerrail
      Contact( "M17.2" )
      Contact( "DB09_TablePos".Req1_Pos )
      I_Contact( "Timer".T10.Q )
      Contact( "Auto" )
      wire#w1
      S_Coil( "M16.3" )
   END_RUNG
   RUNG wire#w1
      R_Coil( "M17.2" )
   END_RUNG
   // the same network as SCL:
   IF "M17.2" AND "DB09_TablePos".Req1_Pos AND NOT "Timer".T10.Q AND "Auto" THEN
       "M16.3" := TRUE;
       "M17.2" := FALSE;
   END_IF;
END_REGION

REGION Network 26: Conveyor cycle: M16.5 Unloading pallet
   RUNG wire#powerrail
      Contact( "M16.3" )
      Contact( "On" )
      wire#w1
      I_Contact( "DB20_DisplaySysdata".dbx38_7 )
      Contact( "Timer".T26.Q )
      Contact( "DB09_TablePos".dbx1_6 )
      Contact( "E43" )
      Contact( "E44" )
      Contact( "DB21_DisplayGeneralData".dbx0_2 )
      Contact( "Auto" )
      wire#w2
      S_Coil( "M16.4" )
   END_RUNG
   RUNG wire#powerrail
      Contact( "M16.5" )
      I_Contact( "E40" )
   END_RUNG wire#w1
   RUNG wire#w2
      R_Coil( "M16.3" )
   END_RUNG
   RUNG wire#w2
      R_Coil( "M16.5" )
   END_RUNG
   // the same network as SCL:
   IF (("M16.3" AND "On") OR ("M16.5" AND NOT "E40")) AND NOT "DB20_DisplaySysdata".dbx38_7 AND "Timer".T26.Q AND "DB09_TablePos".dbx1_6 AND "E43" AND "E44" AND "DB21_DisplayGeneralData".dbx0_2 AND "Auto" THEN
       "M16.4" := TRUE;
   END_IF;
   #_w1 := (("M16.3" AND "On") OR ("M16.5" AND NOT "E40")) AND NOT "DB20_DisplaySysdata".dbx38_7 AND "Timer".T26.Q AND "DB09_TablePos".dbx1_6 AND "E43" AND "E44" AND "DB21_DisplayGeneralData".dbx0_2 AND "Auto";
   IF #_w1 THEN
       "M16.3" := FALSE;
       "M16.5" := FALSE;
   END_IF;
END_REGION

REGION Network 27: Conveyor cycle: M16.3 Unloading pallet
   RUNG wire#powerrail
      Contact( "M16.3" )
      Contact( "Auto" )
      I_Contact( "DB04_Conveyor".dbx4_0 )
      wire#w1
      I_Contact( "E40" )
      wire#w2
      S_Coil( "M16.5" )
   END_RUNG
   RUNG wire#w1
      { S7_Templates := "SrcType := Int" } LT_Contact(in1 := "DB50_Config".Sel6_Selfcenter, in2 := 2)
      I_Contact( "DB21_DisplayGeneralData".dbx0_2 )
   END_RUNG wire#w2
   RUNG wire#w1
      { S7_Templates := "SrcType := Int" } EQ_Contact(in1 := "DB50_Config".Sel6_Selfcenter, in2 := 2)
      Contact( "DB21_DisplayGeneralData".dbx0_5 )
   END_RUNG wire#w2
   RUNG wire#w2
      R_Coil( "M16.3" )
   END_RUNG
   // the same network as SCL:
   IF "M16.3" AND "Auto" AND NOT "DB04_Conveyor".dbx4_0 AND (NOT "E40" OR (("DB50_Config".Sel6_Selfcenter < 2) AND NOT "DB21_DisplayGeneralData".dbx0_2) OR (("DB50_Config".Sel6_Selfcenter = 2) AND "DB21_DisplayGeneralData".dbx0_5)) THEN
       "M16.5" := TRUE;
       "M16.3" := FALSE;
   END_IF;
END_REGION

REGION Network 28: Conveyor cycle: M16.5 Unloading pallet
   RUNG wire#powerrail
      Contact( "M16.5" )
      Contact( "Auto" )
      wire#w1
      Contact( "DB09_TablePos".dbx1_6 )
      wire#w2
      Contact( "E45" )
      wire#w3
      Contact( "Timer".T27.Q )
      wire#w4
      S_Coil( "M17.3" )
   END_RUNG
   RUNG wire#w1
      I_Contact( "DB04_Conveyor".dbx4_3 )
   END_RUNG wire#w2
   RUNG wire#w2
      Contact( "DB21_DisplayGeneralData".dbx0_2 )
   END_RUNG wire#w3
   RUNG wire#w4
      R_Coil( "M16.5" )
   END_RUNG
   RUNG wire#w4
      R_Coil( "M16.3" )
   END_RUNG
   // the same network as SCL:
   IF "M16.5" AND "Auto" AND ("DB09_TablePos".dbx1_6 OR NOT "DB04_Conveyor".dbx4_3) AND ("E45" OR "DB21_DisplayGeneralData".dbx0_2) AND "Timer".T27.Q THEN
       "M17.3" := TRUE;
   END_IF;
   #_w1 := "M16.5" AND "Auto" AND ("DB09_TablePos".dbx1_6 OR NOT "DB04_Conveyor".dbx4_3) AND ("E45" OR "DB21_DisplayGeneralData".dbx0_2) AND "Timer".T27.Q;
   IF #_w1 THEN
       "M16.5" := FALSE;
       "M16.3" := FALSE;
   END_IF;
END_REGION

REGION Network 29: Conveyor cycle: M16.0 Start cycle
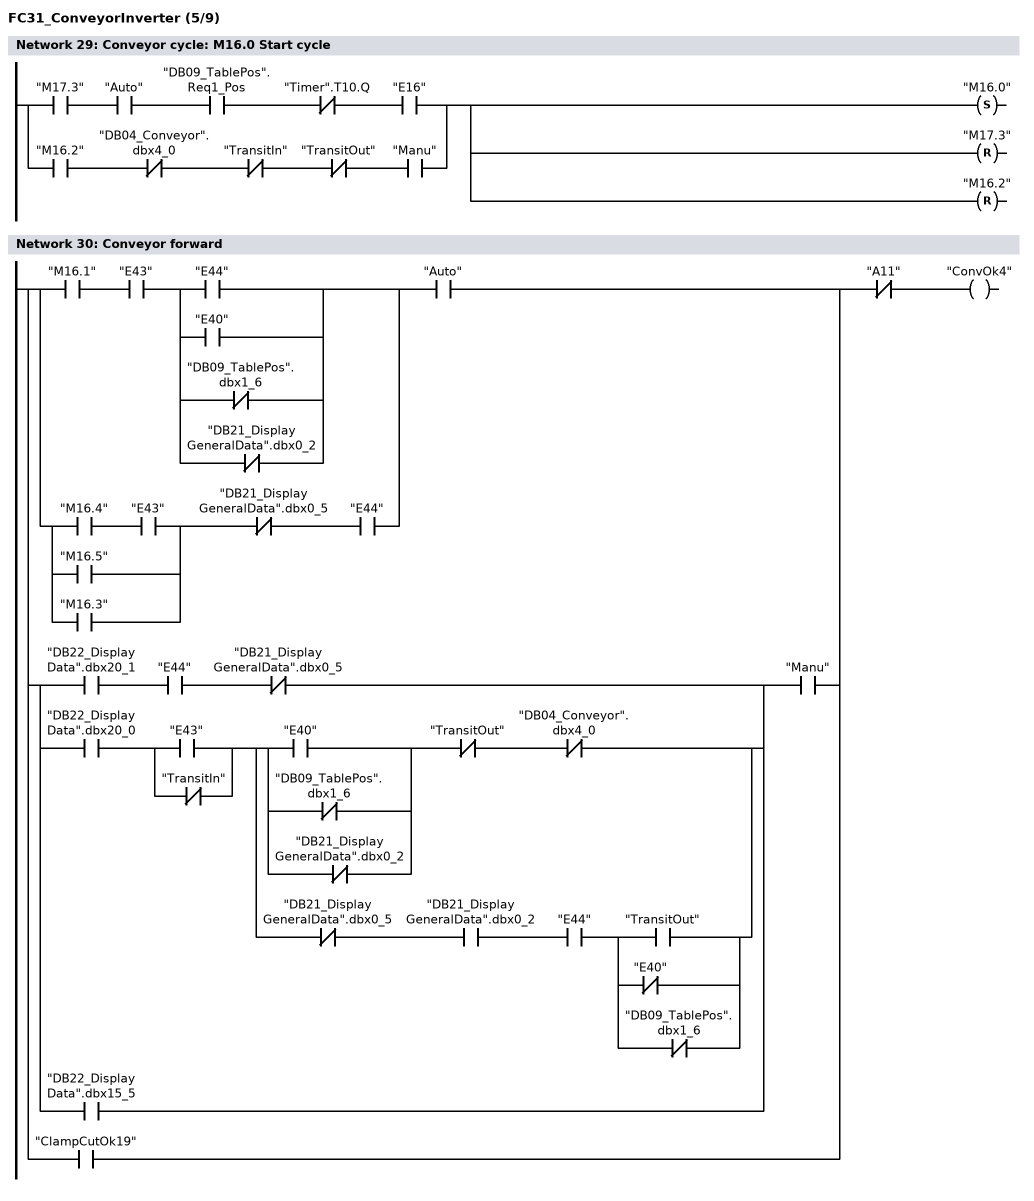
   RUNG wire#powerrail
      Contact( "M17.3" )
      Contact( "Auto" )
      Contact( "DB09_TablePos".Req1_Pos )
      I_Contact( "Timer".T10.Q )
      Contact( "E16" )
      wire#w1
      S_Coil( "M16.0" )
   END_RUNG
   RUNG wire#powerrail
      Contact( "M16.2" )
      I_Contact( "DB04_Conveyor".dbx4_0 )
      I_Contact( "TransitIn" )
      I_Contact( "TransitOut" )
      Contact( "Manu" )
   END_RUNG wire#w1
   RUNG wire#w1
      R_Coil( "M17.3" )
   END_RUNG
   RUNG wire#w1
      R_Coil( "M16.2" )
   END_RUNG
   // the same network as SCL:
   IF ("M17.3" AND "Auto" AND "DB09_TablePos".Req1_Pos AND NOT "Timer".T10.Q AND "E16") OR ("M16.2" AND NOT "DB04_Conveyor".dbx4_0 AND NOT "TransitIn" AND NOT "TransitOut" AND "Manu") THEN
       "M16.0" := TRUE;
   END_IF;
   #_w1 := ("M17.3" AND "Auto" AND "DB09_TablePos".Req1_Pos AND NOT "Timer".T10.Q AND "E16") OR ("M16.2" AND NOT "DB04_Conveyor".dbx4_0 AND NOT "TransitIn" AND NOT "TransitOut" AND "Manu");
   IF #_w1 THEN
       "M17.3" := FALSE;
       "M16.2" := FALSE;
   END_IF;
END_REGION

REGION Network 30: Conveyor forward
   RUNG wire#powerrail
      Contact( "M16.1" )
      Contact( "E43" )
      wire#w1
      Contact( "E44" )
      wire#w2
      Contact( "Auto" )
      wire#w4
      I_Contact( "A11" )
      Coil( "ConvOk4" )
   END_RUNG
   RUNG wire#w1
      Contact( "E40" )
   END_RUNG wire#w2
   RUNG wire#w1
      I_Contact( "DB09_TablePos".dbx1_6 )
   END_RUNG wire#w2
   RUNG wire#w1
      I_Contact( "DB21_DisplayGeneralData".dbx0_2 )
   END_RUNG wire#w2
   RUNG wire#powerrail
      Contact( "M16.4" )
      Contact( "E43" )
      wire#w3
      I_Contact( "DB21_DisplayGeneralData".dbx0_5 )
      Contact( "E44" )
   END_RUNG wire#w2
   RUNG wire#powerrail
      Contact( "M16.5" )
   END_RUNG wire#w3
   RUNG wire#powerrail
      Contact( "M16.3" )
   END_RUNG wire#w3
   RUNG wire#powerrail
      Contact( "DB22_DisplayData".dbx20_1 )
      Contact( "E44" )
      I_Contact( "DB21_DisplayGeneralData".dbx0_5 )
      wire#w5
      Contact( "Manu" )
   END_RUNG wire#w4
   RUNG wire#powerrail
      Contact( "DB22_DisplayData".dbx20_0 )
      wire#w6
      Contact( "E43" )
      wire#w7
      Contact( "E40" )
      wire#w8
      I_Contact( "TransitOut" )
      I_Contact( "DB04_Conveyor".dbx4_0 )
   END_RUNG wire#w5
   RUNG wire#w6
      I_Contact( "TransitIn" )
   END_RUNG wire#w7
   RUNG wire#w7
      I_Contact( "DB09_TablePos".dbx1_6 )
   END_RUNG wire#w8
   RUNG wire#w7
      I_Contact( "DB21_DisplayGeneralData".dbx0_2 )
   END_RUNG wire#w8
   RUNG wire#w7
      I_Contact( "DB21_DisplayGeneralData".dbx0_5 )
      Contact( "DB21_DisplayGeneralData".dbx0_2 )
      Contact( "E44" )
      wire#w9
      Contact( "TransitOut" )
   END_RUNG wire#w5
   RUNG wire#w9
      I_Contact( "E40" )
   END_RUNG wire#w5
   RUNG wire#w9
      I_Contact( "DB09_TablePos".dbx1_6 )
   END_RUNG wire#w5
   RUNG wire#powerrail
      Contact( "DB22_DisplayData".dbx15_5 )
   END_RUNG wire#w5
   RUNG wire#powerrail
      Contact( "ClampCutOk19" )
   END_RUNG wire#w4
   // the same network as SCL:
   "ConvOk4" := (((("M16.1" AND "E43" AND ("E44" OR "E40" OR NOT "DB09_TablePos".dbx1_6 OR NOT "DB21_DisplayGeneralData".dbx0_2)) OR ((("M16.4" AND "E43") OR "M16.5" OR "M16.3") AND NOT "DB21_DisplayGeneralData".dbx0_5 AND "E44")) AND "Auto") OR ((("DB22_DisplayData".dbx20_1 AND "E44" AND NOT "DB21_DisplayGeneralData".dbx0_5) OR ("DB22_DisplayData".dbx20_0 AND ("E43" OR NOT "TransitIn") AND ((("E40" OR NOT "DB09_TablePos".dbx1_6 OR NOT "DB21_DisplayGeneralData".dbx0_2) AND NOT "TransitOut" AND NOT "DB04_Conveyor".dbx4_0) OR (NOT "DB21_DisplayGeneralData".dbx0_5 AND "DB21_DisplayGeneralData".dbx0_2 AND "E44" AND ("TransitOut" OR NOT "E40" OR NOT "DB09_TablePos".dbx1_6)))) OR "DB22_DisplayData".dbx15_5) AND "Manu") OR "ClampCutOk19") AND NOT "A11";
END_REGION

REGION Network 31: ConvOk7: Backward for inverter
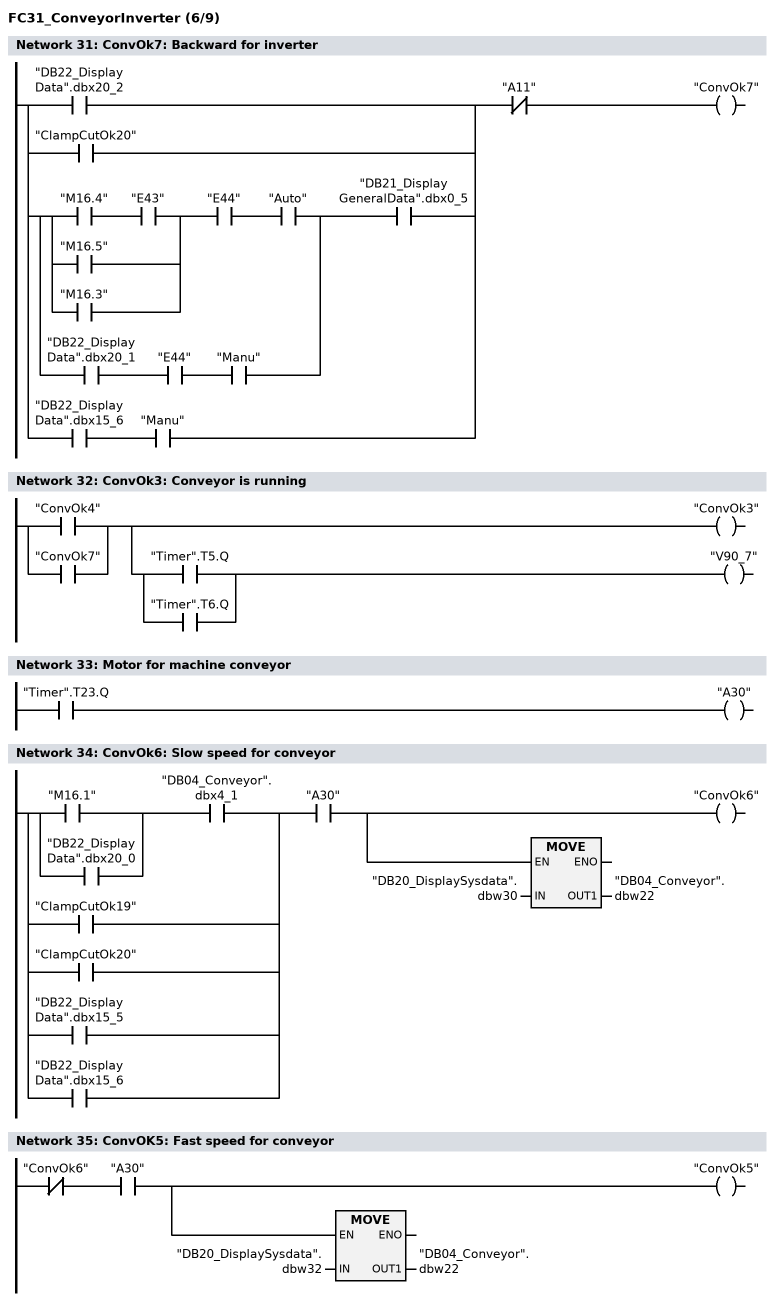
   RUNG wire#powerrail
      Contact( "DB22_DisplayData".dbx20_2 )
      wire#w1
      I_Contact( "A11" )
      Coil( "ConvOk7" )
   END_RUNG
   RUNG wire#powerrail
      Contact( "ClampCutOk20" )
   END_RUNG wire#w1
   RUNG wire#powerrail
      Contact( "M16.4" )
      Contact( "E43" )
      wire#w2
      Contact( "E44" )
      Contact( "Auto" )
      wire#w3
      Contact( "DB21_DisplayGeneralData".dbx0_5 )
   END_RUNG wire#w1
   RUNG wire#powerrail
      Contact( "M16.5" )
   END_RUNG wire#w2
   RUNG wire#powerrail
      Contact( "M16.3" )
   END_RUNG wire#w2
   RUNG wire#powerrail
      Contact( "DB22_DisplayData".dbx20_1 )
      Contact( "E44" )
      Contact( "Manu" )
   END_RUNG wire#w3
   RUNG wire#powerrail
      Contact( "DB22_DisplayData".dbx15_6 )
      Contact( "Manu" )
   END_RUNG wire#w1
   // the same network as SCL:
   "ConvOk7" := ("DB22_DisplayData".dbx20_2 OR "ClampCutOk20" OR ((((("M16.4" AND "E43") OR "M16.5" OR "M16.3") AND "E44" AND "Auto") OR ("DB22_DisplayData".dbx20_1 AND "E44" AND "Manu")) AND "DB21_DisplayGeneralData".dbx0_5) OR ("DB22_DisplayData".dbx15_6 AND "Manu")) AND NOT "A11";
END_REGION

REGION Network 32: ConvOk3: Conveyor is running
   RUNG wire#powerrail
      Contact( "ConvOk4" )
      wire#w1
      Coil( "ConvOk3" )
   END_RUNG
   RUNG wire#powerrail
      Contact( "ConvOk7" )
   END_RUNG wire#w1
   RUNG wire#w1
      Contact( "Timer".T5.Q )
      wire#w2
      Coil( "V90_7" )
   END_RUNG
   RUNG wire#w1
      Contact( "Timer".T6.Q )
   END_RUNG wire#w2
   // the same network as SCL:
   "ConvOk3" := "ConvOk4" OR "ConvOk7";
   "V90_7" := "ConvOk3" AND ("Timer".T5.Q OR "Timer".T6.Q);
END_REGION

REGION Network 33: Motor for machine conveyor
   RUNG wire#powerrail
      Contact( "Timer".T23.Q )
      Coil( "A30" )
   END_RUNG
   // the same network as SCL:
   "A30" := "Timer".T23.Q;
END_REGION

REGION Network 34: ConvOk6: Slow speed for conveyor
   RUNG wire#powerrail
      Contact( "M16.1" )
      wire#w1
      Contact( "DB04_Conveyor".dbx4_1 )
      wire#w2
      Contact( "A30" )
      wire#w3
      Coil( "ConvOk6" )
   END_RUNG
   RUNG wire#powerrail
      Contact( "DB22_DisplayData".dbx20_0 )
   END_RUNG wire#w1
   RUNG wire#powerrail
      Contact( "ClampCutOk19" )
   END_RUNG wire#w2
   RUNG wire#powerrail
      Contact( "ClampCutOk20" )
   END_RUNG wire#w2
   RUNG wire#powerrail
      Contact( "DB22_DisplayData".dbx15_5 )
   END_RUNG wire#w2
   RUNG wire#powerrail
      Contact( "DB22_DisplayData".dbx15_6 )
   END_RUNG wire#w2
   RUNG wire#w3
      { S7_GenerateENO := "TRUE" } Move(in := "DB20_DisplaySysdata".dbw30, out1 => "DB04_Conveyor".dbw22)
   END_RUNG
   // the same network as SCL:
   "ConvOk6" := ((("M16.1" OR "DB22_DisplayData".dbx20_0) AND "DB04_Conveyor".dbx4_1) OR "ClampCutOk19" OR "ClampCutOk20" OR "DB22_DisplayData".dbx15_5 OR "DB22_DisplayData".dbx15_6) AND "A30";
   IF "ConvOk6" THEN "DB04_Conveyor".dbw22 := "DB20_DisplaySysdata".dbw30; END_IF;
END_REGION

REGION Network 35: ConvOK5: Fast speed for conveyor
   RUNG wire#powerrail
      I_Contact( "ConvOk6" )
      Contact( "A30" )
      wire#w1
      Coil( "ConvOk5" )
   END_RUNG
   RUNG wire#w1
      { S7_GenerateENO := "TRUE" } Move(in := "DB20_DisplaySysdata".dbw32, out1 => "DB04_Conveyor".dbw22)
   END_RUNG
   // the same network as SCL:
   "ConvOk5" := NOT "ConvOk6" AND "A30";
   IF "ConvOk5" THEN "DB04_Conveyor".dbw22 := "DB20_DisplaySysdata".dbw32; END_IF;
END_REGION

REGION Network 36: rotation inverter: Support for speed selection
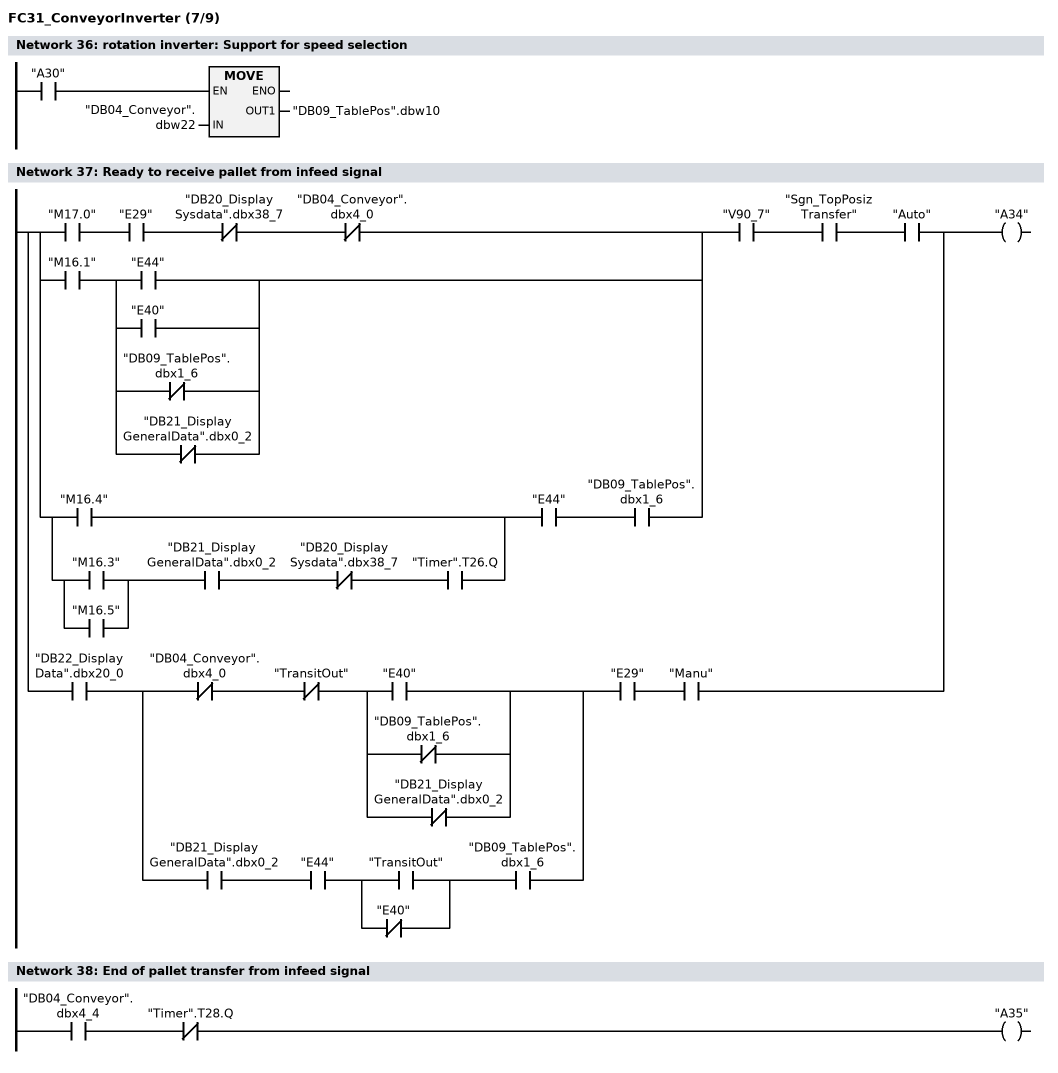
   RUNG wire#powerrail
      Contact( "A30" )
      { S7_GenerateENO := "TRUE" } Move(in := "DB04_Conveyor".dbw22, out1 => "DB09_TablePos".dbw10)
   END_RUNG
   // the same network as SCL:
   IF "A30" THEN "DB09_TablePos".dbw10 := "DB04_Conveyor".dbw22; END_IF;
END_REGION

REGION Network 37: Ready to receive pallet from infeed signal
   RUNG wire#powerrail
      Contact( "M17.0" )
      Contact( "E29" )
      I_Contact( "DB20_DisplaySysdata".dbx38_7 )
      I_Contact( "DB04_Conveyor".dbx4_0 )
      wire#w1
      Contact( "V90_7" )
      Contact( "Sgn_TopPosizTransfer" )
      Contact( "Auto" )
      wire#w5
      Coil( "A34" )
   END_RUNG
   RUNG wire#powerrail
      Contact( "M16.1" )
      wire#w2
      Contact( "E44" )
   END_RUNG wire#w1
   RUNG wire#w2
      Contact( "E40" )
   END_RUNG wire#w1
   RUNG wire#w2
      I_Contact( "DB09_TablePos".dbx1_6 )
   END_RUNG wire#w1
   RUNG wire#w2
      I_Contact( "DB21_DisplayGeneralData".dbx0_2 )
   END_RUNG wire#w1
   RUNG wire#powerrail
      Contact( "M16.4" )
      wire#w3
      Contact( "E44" )
      Contact( "DB09_TablePos".dbx1_6 )
   END_RUNG wire#w1
   RUNG wire#powerrail
      Contact( "M16.3" )
      wire#w4
      Contact( "DB21_DisplayGeneralData".dbx0_2 )
      I_Contact( "DB20_DisplaySysdata".dbx38_7 )
      Contact( "Timer".T26.Q )
   END_RUNG wire#w3
   RUNG wire#powerrail
      Contact( "M16.5" )
   END_RUNG wire#w4
   RUNG wire#powerrail
      Contact( "DB22_DisplayData".dbx20_0 )
      wire#w6
      I_Contact( "DB04_Conveyor".dbx4_0 )
      I_Contact( "TransitOut" )
      wire#w7
      Contact( "E40" )
      wire#w8
      Contact( "E29" )
      Contact( "Manu" )
   END_RUNG wire#w5
   RUNG wire#w7
      I_Contact( "DB09_TablePos".dbx1_6 )
   END_RUNG wire#w8
   RUNG wire#w7
      I_Contact( "DB21_DisplayGeneralData".dbx0_2 )
   END_RUNG wire#w8
   RUNG wire#w6
      Contact( "DB21_DisplayGeneralData".dbx0_2 )
      Contact( "E44" )
      wire#w9
      Contact( "TransitOut" )
      wire#w10
      Contact( "DB09_TablePos".dbx1_6 )
   END_RUNG wire#w8
   RUNG wire#w9
      I_Contact( "E40" )
   END_RUNG wire#w10
   // the same network as SCL:
   "A34" := ((("M17.0" AND "E29" AND NOT "DB20_DisplaySysdata".dbx38_7 AND NOT "DB04_Conveyor".dbx4_0) OR ("M16.1" AND ("E44" OR "E40" OR NOT "DB09_TablePos".dbx1_6 OR NOT "DB21_DisplayGeneralData".dbx0_2)) OR (("M16.4" OR (("M16.3" OR "M16.5") AND "DB21_DisplayGeneralData".dbx0_2 AND NOT "DB20_DisplaySysdata".dbx38_7 AND "Timer".T26.Q)) AND "E44" AND "DB09_TablePos".dbx1_6)) AND "V90_7" AND "Sgn_TopPosizTransfer" AND "Auto") OR ("DB22_DisplayData".dbx20_0 AND ((NOT "DB04_Conveyor".dbx4_0 AND NOT "TransitOut" AND ("E40" OR NOT "DB09_TablePos".dbx1_6 OR NOT "DB21_DisplayGeneralData".dbx0_2)) OR ("DB21_DisplayGeneralData".dbx0_2 AND "E44" AND ("TransitOut" OR NOT "E40") AND "DB09_TablePos".dbx1_6)) AND "E29" AND "Manu");
END_REGION

REGION Network 38: End of pallet transfer from infeed signal
   RUNG wire#powerrail
      Contact( "DB04_Conveyor".dbx4_4 )
      I_Contact( "Timer".T28.Q )
      Coil( "A35" )
   END_RUNG
   // the same network as SCL:
   "A35" := "DB04_Conveyor".dbx4_4 AND NOT "Timer".T28.Q;
END_REGION

REGION Network 39: Pallet ready for outfeed signal
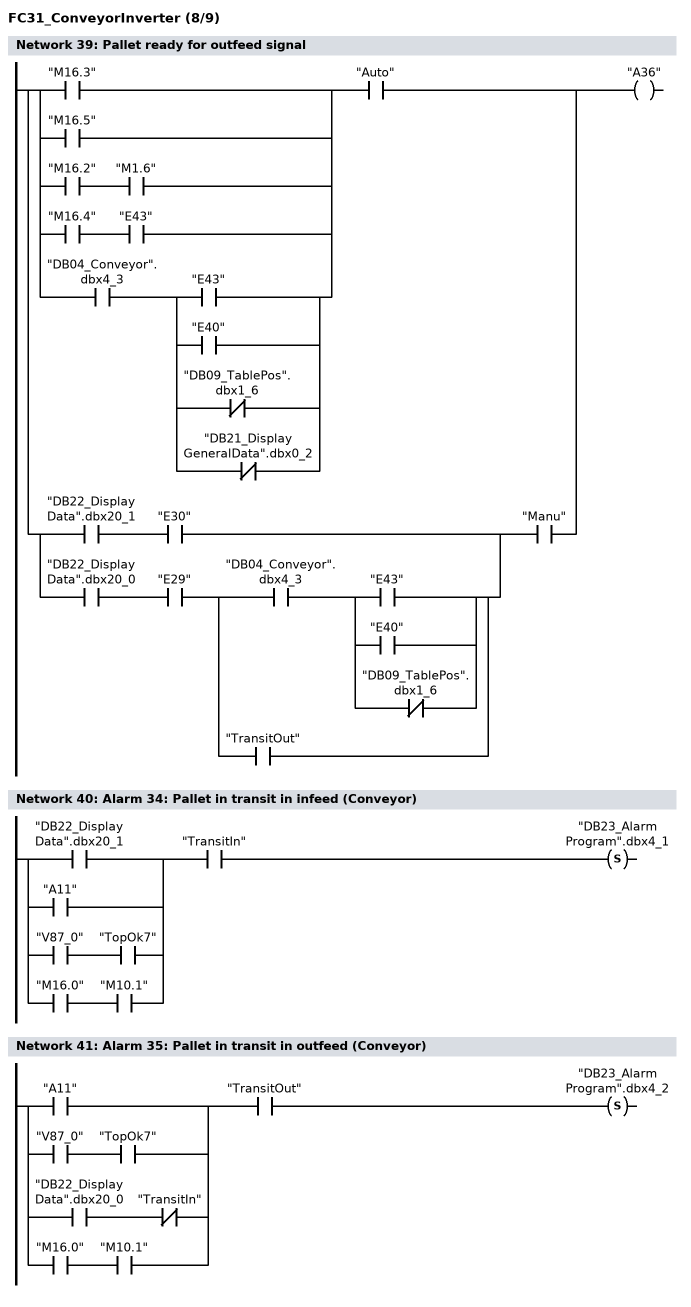
   RUNG wire#powerrail
      Contact( "M16.3" )
      wire#w1
      Contact( "Auto" )
      wire#w3
      Coil( "A36" )
   END_RUNG
   RUNG wire#powerrail
      Contact( "M16.5" )
   END_RUNG wire#w1
   RUNG wire#powerrail
      Contact( "M16.2" )
      Contact( "M1.6" )
   END_RUNG wire#w1
   RUNG wire#powerrail
      Contact( "M16.4" )
      Contact( "E43" )
   END_RUNG wire#w1
   RUNG wire#powerrail
      Contact( "DB04_Conveyor".dbx4_3 )
      wire#w2
      Contact( "E43" )
   END_RUNG wire#w1
   RUNG wire#w2
      Contact( "E40" )
   END_RUNG wire#w1
   RUNG wire#w2
      I_Contact( "DB09_TablePos".dbx1_6 )
   END_RUNG wire#w1
   RUNG wire#w2
      I_Contact( "DB21_DisplayGeneralData".dbx0_2 )
   END_RUNG wire#w1
   RUNG wire#powerrail
      Contact( "DB22_DisplayData".dbx20_1 )
      Contact( "E30" )
      wire#w4
      Contact( "Manu" )
   END_RUNG wire#w3
   RUNG wire#powerrail
      Contact( "DB22_DisplayData".dbx20_0 )
      Contact( "E29" )
      wire#w5
      Contact( "DB04_Conveyor".dbx4_3 )
      wire#w6
      Contact( "E43" )
   END_RUNG wire#w4
   RUNG wire#w6
      Contact( "E40" )
   END_RUNG wire#w4
   RUNG wire#w6
      I_Contact( "DB09_TablePos".dbx1_6 )
   END_RUNG wire#w4
   RUNG wire#w5
      Contact( "TransitOut" )
   END_RUNG wire#w4
   // the same network as SCL:
   "A36" := (("M16.3" OR "M16.5" OR ("M16.2" AND "M1.6") OR ("M16.4" AND "E43") OR ("DB04_Conveyor".dbx4_3 AND ("E43" OR "E40" OR NOT "DB09_TablePos".dbx1_6 OR NOT "DB21_DisplayGeneralData".dbx0_2))) AND "Auto") OR ((("DB22_DisplayData".dbx20_1 AND "E30") OR ("DB22_DisplayData".dbx20_0 AND "E29" AND (("DB04_Conveyor".dbx4_3 AND ("E43" OR "E40" OR NOT "DB09_TablePos".dbx1_6)) OR "TransitOut"))) AND "Manu");
END_REGION

REGION Network 40: Alarm 34: Pallet in transit in infeed (Conveyor)
   RUNG wire#powerrail
      Contact( "DB22_DisplayData".dbx20_1 )
      wire#w1
      Contact( "TransitIn" )
      S_Coil( "DB23_AlarmProgram".dbx4_1 )
   END_RUNG
   RUNG wire#powerrail
      Contact( "A11" )
   END_RUNG wire#w1
   RUNG wire#powerrail
      Contact( "V87_0" )
      Contact( "TopOk7" )
   END_RUNG wire#w1
   RUNG wire#powerrail
      Contact( "M16.0" )
      Contact( "M10.1" )
   END_RUNG wire#w1
   // the same network as SCL:
   IF ("DB22_DisplayData".dbx20_1 OR "A11" OR ("V87_0" AND "TopOk7") OR ("M16.0" AND "M10.1")) AND "TransitIn" THEN
       "DB23_AlarmProgram".dbx4_1 := TRUE;
   END_IF;
END_REGION

REGION Network 41: Alarm 35: Pallet in transit in outfeed (Conveyor)
   RUNG wire#powerrail
      Contact( "A11" )
      wire#w1
      Contact( "TransitOut" )
      S_Coil( "DB23_AlarmProgram".dbx4_2 )
   END_RUNG
   RUNG wire#powerrail
      Contact( "V87_0" )
      Contact( "TopOk7" )
   END_RUNG wire#w1
   RUNG wire#powerrail
      Contact( "DB22_DisplayData".dbx20_0 )
      I_Contact( "TransitIn" )
   END_RUNG wire#w1
   RUNG wire#powerrail
      Contact( "M16.0" )
      Contact( "M10.1" )
   END_RUNG wire#w1
   // the same network as SCL:
   IF ("A11" OR ("V87_0" AND "TopOk7") OR ("DB22_DisplayData".dbx20_0 AND NOT "TransitIn") OR ("M16.0" AND "M10.1")) AND "TransitOut" THEN
       "DB23_AlarmProgram".dbx4_2 := TRUE;
   END_IF;
END_REGION

REGION Network 42: Alarm 39: Technoplat table not in load phase
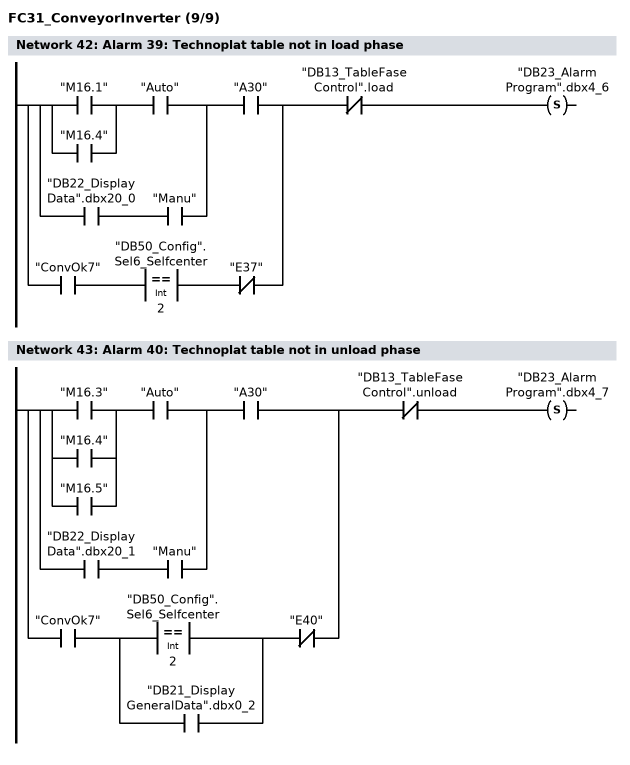
   RUNG wire#powerrail
      Contact( "M16.1" )
      wire#w1
      Contact( "Auto" )
      wire#w2
      Contact( "A30" )
      wire#w3
      I_Contact( "DB13_TableFaseControl".load )
      S_Coil( "DB23_AlarmProgram".dbx4_6 )
   END_RUNG
   RUNG wire#powerrail
      Contact( "M16.4" )
   END_RUNG wire#w1
   RUNG wire#powerrail
      Contact( "DB22_DisplayData".dbx20_0 )
      Contact( "Manu" )
   END_RUNG wire#w2
   RUNG wire#powerrail
      Contact( "ConvOk7" )
      { S7_Templates := "SrcType := Int" } EQ_Contact(in1 := "DB50_Config".Sel6_Selfcenter, in2 := 2)
      I_Contact( "E37" )
   END_RUNG wire#w3
   // the same network as SCL:
   IF ((((("M16.1" OR "M16.4") AND "Auto") OR ("DB22_DisplayData".dbx20_0 AND "Manu")) AND "A30") OR ("ConvOk7" AND ("DB50_Config".Sel6_Selfcenter = 2) AND NOT "E37")) AND NOT "DB13_TableFaseControl".load THEN
       "DB23_AlarmProgram".dbx4_6 := TRUE;
   END_IF;
END_REGION

REGION Network 43: Alarm 40: Technoplat table not in unload phase
   RUNG wire#powerrail
      Contact( "M16.3" )
      wire#w1
      Contact( "Auto" )
      wire#w2
      Contact( "A30" )
      wire#w3
      I_Contact( "DB13_TableFaseControl".unload )
      S_Coil( "DB23_AlarmProgram".dbx4_7 )
   END_RUNG
   RUNG wire#powerrail
      Contact( "M16.4" )
   END_RUNG wire#w1
   RUNG wire#powerrail
      Contact( "M16.5" )
   END_RUNG wire#w1
   RUNG wire#powerrail
      Contact( "DB22_DisplayData".dbx20_1 )
      Contact( "Manu" )
   END_RUNG wire#w2
   RUNG wire#powerrail
      Contact( "ConvOk7" )
      wire#w4
      { S7_Templates := "SrcType := Int" } EQ_Contact(in1 := "DB50_Config".Sel6_Selfcenter, in2 := 2)
      wire#w5
      I_Contact( "E40" )
   END_RUNG wire#w3
   RUNG wire#w4
      Contact( "DB21_DisplayGeneralData".dbx0_2 )
   END_RUNG wire#w5
   // the same network as SCL:
   IF ((((("M16.3" OR "M16.4" OR "M16.5") AND "Auto") OR ("DB22_DisplayData".dbx20_1 AND "Manu")) AND "A30") OR ("ConvOk7" AND (("DB50_Config".Sel6_Selfcenter = 2) OR "DB21_DisplayGeneralData".dbx0_2) AND NOT "E40")) AND NOT "DB13_TableFaseControl".unload THEN
       "DB23_AlarmProgram".dbx4_7 := TRUE;
   END_IF;
END_REGION
END_FUNCTION

FUNCTION "FC37_MultiprogramSignal" : Void   // FC37, LAD
TITLE = Multiprogram with program selection by external signal
{ S7_Optimized_Access := 'FALSE' }
AUTHOR : Robopac
VERSION : 0.0
// stored: AutoNumber false, IsIECCheckEnabled false, SetENOAutomatically false, UDAEnableTagReadback false
   VAR_TEMP   // added for the SCL form of the ladder/FBD networks
      _w1 : Bool;
   END_VAR
BEGIN

REGION Network 1
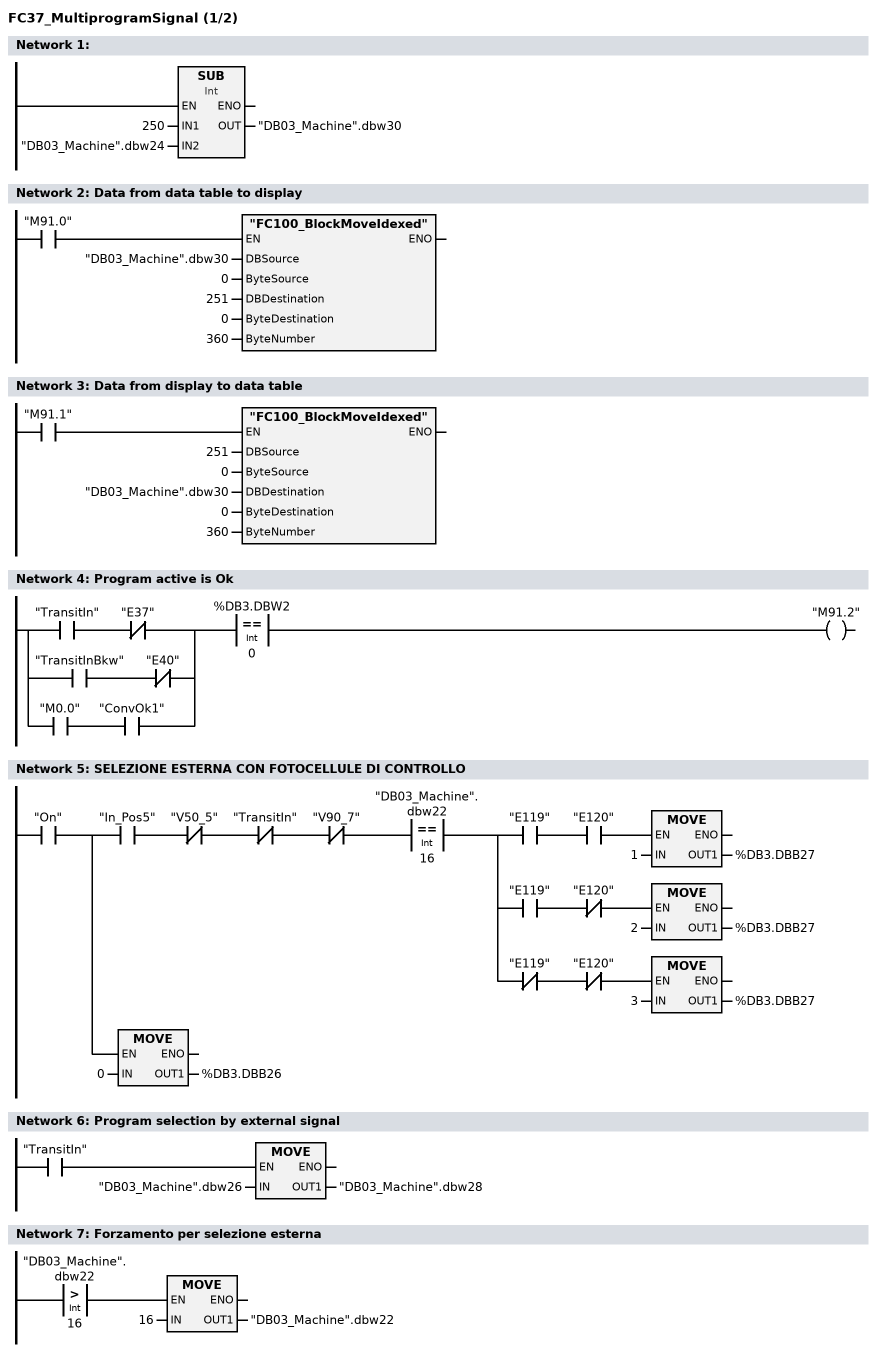
   RUNG wire#powerrail
      { S7_Templates := "SrcType := Int"; S7_GenerateENO := "TRUE" } Sub(in1 := 250, in2 := "DB03_Machine".dbw24, out => "DB03_Machine".dbw30)
   END_RUNG
   // the same network as SCL:
   "DB03_Machine".dbw30 := 250 - "DB03_Machine".dbw24;
END_REGION

REGION Network 2: Data from data table to display
   RUNG wire#powerrail
      Contact( "M91.0" )
      "FC100_BlockMoveIdexed"(DBSource := "DB03_Machine".dbw30, ByteSource := 0, DBDestination := 251, ByteDestination := 0, ByteNumber := 360)
   END_RUNG
   // the same network as SCL:
   IF "M91.0" THEN
       "FC100_BlockMoveIdexed"(DBSource := "DB03_Machine".dbw30,
                               ByteSource := 0,
                               DBDestination := 251,
                               ByteDestination := 0,
                               ByteNumber := 360);
   END_IF;
END_REGION

REGION Network 3: Data from display to data table
   RUNG wire#powerrail
      Contact( "M91.1" )
      "FC100_BlockMoveIdexed"(DBSource := 251, ByteSource := 0, DBDestination := "DB03_Machine".dbw30, ByteDestination := 0, ByteNumber := 360)
   END_RUNG
   // the same network as SCL:
   IF "M91.1" THEN
       "FC100_BlockMoveIdexed"(DBSource := 251,
                               ByteSource := 0,
                               DBDestination := "DB03_Machine".dbw30,
                               ByteDestination := 0,
                               ByteNumber := 360);
   END_IF;
END_REGION

REGION Network 4: Program active is Ok
   RUNG wire#powerrail
      Contact( "TransitIn" )
      I_Contact( "E37" )
      wire#w1
      { S7_Templates := "SrcType := Int" } EQ_Contact(in1 := %DB3.DBW2, in2 := 0)
      Coil( "M91.2" )
   END_RUNG
   RUNG wire#powerrail
      Contact( "TransitInBkw" )
      I_Contact( "E40" )
   END_RUNG wire#w1
   RUNG wire#powerrail
      Contact( "M0.0" )
      Contact( "ConvOk1" )
   END_RUNG wire#w1
   // the same network as SCL:
   "M91.2" := (("TransitIn" AND NOT "E37") OR ("TransitInBkw" AND NOT "E40") OR ("M0.0" AND "ConvOk1")) AND (%DB3.DBW2 = 0);
END_REGION

REGION Network 5: SELEZIONE ESTERNA CON FOTOCELLULE DI CONTROLLO
   RUNG wire#powerrail
      Contact( "On" )
      wire#w1
      Contact( "In_Pos5" )
      I_Contact( "V50_5" )
      I_Contact( "TransitIn" )
      I_Contact( "V90_7" )
      { S7_Templates := "SrcType := Int" } EQ_Contact(in1 := "DB03_Machine".dbw22, in2 := 16)
      wire#w2
      Contact( "E119" )
      Contact( "E120" )
      Move(in := 1, out1 => %DB3.DBB27)
   END_RUNG
   RUNG wire#w2
      Contact( "E119" )
      I_Contact( "E120" )
      Move(in := 2, out1 => %DB3.DBB27)
   END_RUNG
   RUNG wire#w2
      I_Contact( "E119" )
      I_Contact( "E120" )
      Move(in := 3, out1 => %DB3.DBB27)
   END_RUNG
   RUNG wire#w1
      { S7_GenerateENO := "TRUE" } Move(in := 0, out1 => %DB3.DBB26)
   END_RUNG
   // the same network as SCL:
   #_w1 := "On" AND "In_Pos5" AND NOT "V50_5" AND NOT "TransitIn" AND NOT "V90_7" AND ("DB03_Machine".dbw22 = 16);
   IF #_w1 AND "E119" AND "E120" THEN %DB3.DBB27 := 1; END_IF;
   IF #_w1 AND "E119" AND NOT "E120" THEN %DB3.DBB27 := 2; END_IF;
   IF #_w1 AND NOT "E119" AND NOT "E120" THEN %DB3.DBB27 := 3; END_IF;
   IF "On" THEN %DB3.DBB26 := 0; END_IF;
END_REGION

REGION Network 6: Program selection by external signal
   RUNG wire#powerrail
      Contact( "TransitIn" )
      { S7_GenerateENO := "TRUE" } Move(in := "DB03_Machine".dbw26, out1 => "DB03_Machine".dbw28)
   END_RUNG
   // the same network as SCL:
   IF "TransitIn" THEN "DB03_Machine".dbw28 := "DB03_Machine".dbw26; END_IF;
END_REGION

REGION Network 7: Forzamento per selezione esterna
   RUNG wire#powerrail
      { S7_Templates := "SrcType := Int" } GT_Contact(in1 := "DB03_Machine".dbw22, in2 := 16)
      { S7_GenerateENO := "TRUE" } Move(in := 16, out1 => "DB03_Machine".dbw22)
   END_RUNG
   // the same network as SCL:
   IF "DB03_Machine".dbw22 > 16 THEN "DB03_Machine".dbw22 := 16; END_IF;
END_REGION

REGION Network 8: Program selection by display
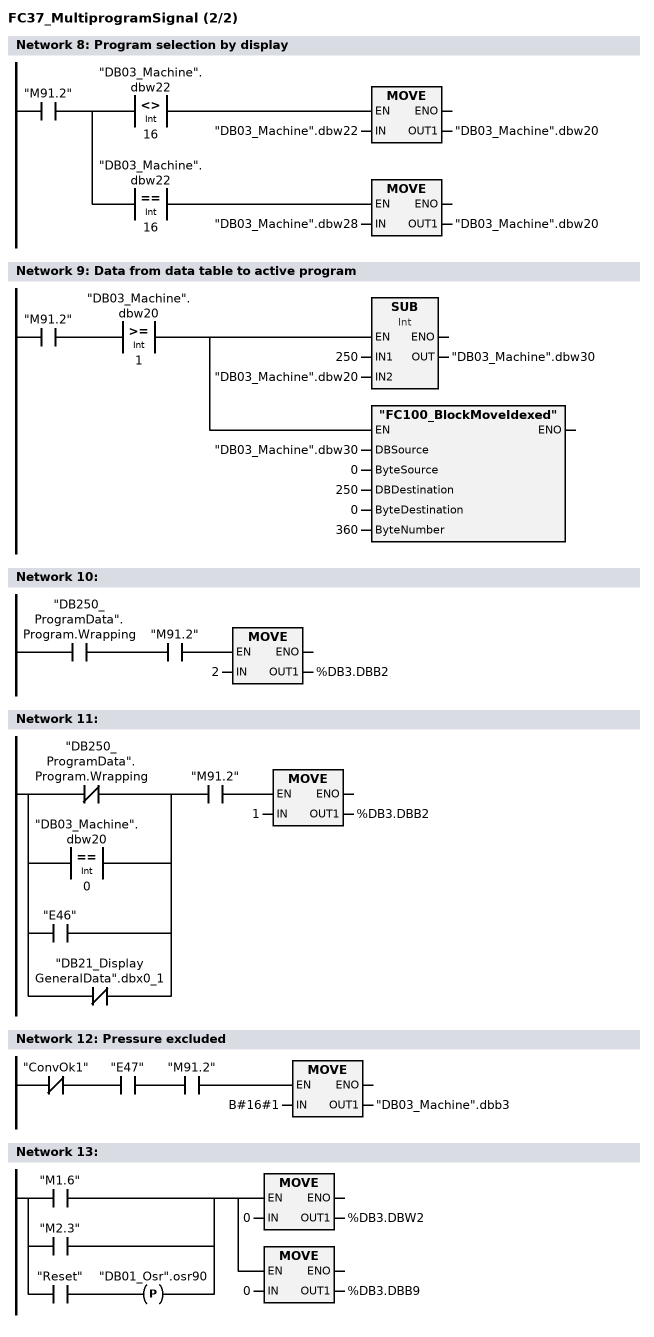
   RUNG wire#powerrail
      Contact( "M91.2" )
      wire#w1
      { S7_Templates := "SrcType := Int" } NE_Contact(in1 := "DB03_Machine".dbw22, in2 := 16)
      { S7_GenerateENO := "TRUE" } Move(in := "DB03_Machine".dbw22, out1 => "DB03_Machine".dbw20)
   END_RUNG
   RUNG wire#w1
      { S7_Templates := "SrcType := Int" } EQ_Contact(in1 := "DB03_Machine".dbw22, in2 := 16)
      { S7_GenerateENO := "TRUE" } Move(in := "DB03_Machine".dbw28, out1 => "DB03_Machine".dbw20)
   END_RUNG
   // the same network as SCL:
   IF "M91.2" AND ("DB03_Machine".dbw22 <> 16) THEN "DB03_Machine".dbw20 := "DB03_Machine".dbw22; END_IF;
   IF "M91.2" AND ("DB03_Machine".dbw22 = 16) THEN "DB03_Machine".dbw20 := "DB03_Machine".dbw28; END_IF;
END_REGION

REGION Network 9: Data from data table to active program
   RUNG wire#powerrail
      Contact( "M91.2" )
      { S7_Templates := "SrcType := Int" } GE_Contact(in1 := "DB03_Machine".dbw20, in2 := 1)
      wire#w1
      { S7_Templates := "SrcType := Int"; S7_GenerateENO := "TRUE" } Sub(in1 := 250, in2 := "DB03_Machine".dbw20, out => "DB03_Machine".dbw30)
   END_RUNG
   RUNG wire#w1
      "FC100_BlockMoveIdexed"(DBSource := "DB03_Machine".dbw30, ByteSource := 0, DBDestination := 250, ByteDestination := 0, ByteNumber := 360)
   END_RUNG
   // the same network as SCL:
   IF "M91.2" AND ("DB03_Machine".dbw20 >= 1) THEN
       "DB03_Machine".dbw30 := 250 - "DB03_Machine".dbw20;
       "FC100_BlockMoveIdexed"(DBSource := "DB03_Machine".dbw30,
                               ByteSource := 0,
                               DBDestination := 250,
                               ByteDestination := 0,
                               ByteNumber := 360);
   END_IF;
END_REGION

REGION Network 10
   RUNG wire#powerrail
      Contact( "DB250_ProgramData".Program.Wrapping )
      Contact( "M91.2" )
      { S7_GenerateENO := "TRUE" } Move(in := 2, out1 => %DB3.DBB2)
   END_RUNG
   // the same network as SCL:
   IF "DB250_ProgramData".Program.Wrapping AND "M91.2" THEN %DB3.DBB2 := 2; END_IF;
END_REGION

REGION Network 11
   RUNG wire#powerrail
      I_Contact( "DB250_ProgramData".Program.Wrapping )
      wire#w1
      Contact( "M91.2" )
      { S7_GenerateENO := "TRUE" } Move(in := 1, out1 => %DB3.DBB2)
   END_RUNG
   RUNG wire#powerrail
      { S7_Templates := "SrcType := Int" } EQ_Contact(in1 := "DB03_Machine".dbw20, in2 := 0)
   END_RUNG wire#w1
   RUNG wire#powerrail
      Contact( "E46" )
   END_RUNG wire#w1
   RUNG wire#powerrail
      I_Contact( "DB21_DisplayGeneralData".dbx0_1 )
   END_RUNG wire#w1
   // the same network as SCL:
   IF (NOT "DB250_ProgramData".Program.Wrapping OR ("DB03_Machine".dbw20 = 0) OR "E46" OR NOT "DB21_DisplayGeneralData".dbx0_1) AND "M91.2" THEN
       %DB3.DBB2 := 1;
   END_IF;
END_REGION

REGION Network 12: Pressure excluded
   RUNG wire#powerrail
      I_Contact( "ConvOk1" )
      Contact( "E47" )
      Contact( "M91.2" )
      { S7_GenerateENO := "TRUE" } Move(in := B#16#1, out1 => "DB03_Machine".dbb3)
   END_RUNG
   // the same network as SCL:
   IF NOT "ConvOk1" AND "E47" AND "M91.2" THEN "DB03_Machine".dbb3 := B#16#1; END_IF;
END_REGION

REGION Network 13
   RUNG wire#powerrail
      Contact( "M1.6" )
      wire#w1
      { S7_GenerateENO := "TRUE" } Move(in := 0, out1 => %DB3.DBW2)
   END_RUNG
   RUNG wire#powerrail
      Contact( "M2.3" )
   END_RUNG wire#w1
   RUNG wire#powerrail
      Contact( "Reset" )
      P_Trig( "DB01_Osr".osr90 )
   END_RUNG wire#w1
   RUNG wire#w1
      { S7_GenerateENO := "TRUE" } Move(in := 0, out1 => %DB3.DBB9)
   END_RUNG
   // the same network as SCL:
   #_w1 := "Reset" AND NOT "DB01_Osr".osr90;   // rising edge
   "DB01_Osr".osr90 := "Reset";
   IF "M1.6" OR "M2.3" OR #_w1 THEN
       %DB3.DBW2 := 0;
       %DB3.DBB9 := 0;
   END_IF;
END_REGION
END_FUNCTION

FUNCTION "FC39_DisplaySiemensTP" : Void   // FC39, LAD
TITLE = Display Siemens TP177 management
{ S7_Optimized_Access := 'FALSE' }
AUTHOR : Robopac
VERSION : 0.0
// stored: AutoNumber false, IsIECCheckEnabled false, SetENOAutomatically false, UDAEnableTagReadback false
   VAR_TEMP
      TempInt : Int;
   END_VAR
   VAR_TEMP   // added for the SCL form of the ladder/FBD networks
      _w1 : Bool;
      _w2 : Bool;
      _w3 : Bool;
      _w4 : Bool;
      _w5 : Bool;
      _w6 : Bool;
   END_VAR
BEGIN

REGION Network 1: Manual(Toggle bit): Pressure plate upward/downward (Helix)
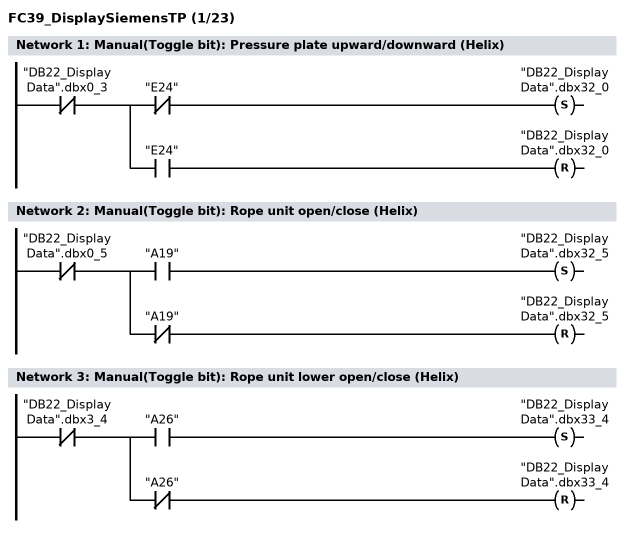
   RUNG wire#powerrail
      I_Contact( "DB22_DisplayData".dbx0_3 )
      wire#w1
      I_Contact( "E24" )
      S_Coil( "DB22_DisplayData".dbx32_0 )
   END_RUNG
   RUNG wire#w1
      Contact( "E24" )
      R_Coil( "DB22_DisplayData".dbx32_0 )
   END_RUNG
   // the same network as SCL:
   #_w1 := NOT "DB22_DisplayData".dbx0_3;
   IF #_w1 AND NOT "E24" THEN "DB22_DisplayData".dbx32_0 := TRUE; END_IF;
   IF #_w1 AND "E24" THEN "DB22_DisplayData".dbx32_0 := FALSE; END_IF;
END_REGION

REGION Network 2: Manual(Toggle bit): Rope unit open/close (Helix)
   RUNG wire#powerrail
      I_Contact( "DB22_DisplayData".dbx0_5 )
      wire#w1
      Contact( "A19" )
      S_Coil( "DB22_DisplayData".dbx32_5 )
   END_RUNG
   RUNG wire#w1
      I_Contact( "A19" )
      R_Coil( "DB22_DisplayData".dbx32_5 )
   END_RUNG
   // the same network as SCL:
   #_w1 := NOT "DB22_DisplayData".dbx0_5;
   IF #_w1 AND "A19" THEN "DB22_DisplayData".dbx32_5 := TRUE; END_IF;
   IF #_w1 AND NOT "A19" THEN "DB22_DisplayData".dbx32_5 := FALSE; END_IF;
END_REGION

REGION Network 3: Manual(Toggle bit): Rope unit lower open/close (Helix)
   RUNG wire#powerrail
      I_Contact( "DB22_DisplayData".dbx3_4 )
      wire#w1
      Contact( "A26" )
      S_Coil( "DB22_DisplayData".dbx33_4 )
   END_RUNG
   RUNG wire#w1
      I_Contact( "A26" )
      R_Coil( "DB22_DisplayData".dbx33_4 )
   END_RUNG
   // the same network as SCL:
   #_w1 := NOT "DB22_DisplayData".dbx3_4;
   IF #_w1 AND "A26" THEN "DB22_DisplayData".dbx33_4 := TRUE; END_IF;
   IF #_w1 AND NOT "A26" THEN "DB22_DisplayData".dbx33_4 := FALSE; END_IF;
END_REGION

REGION Network 4: Manual operation for Helix
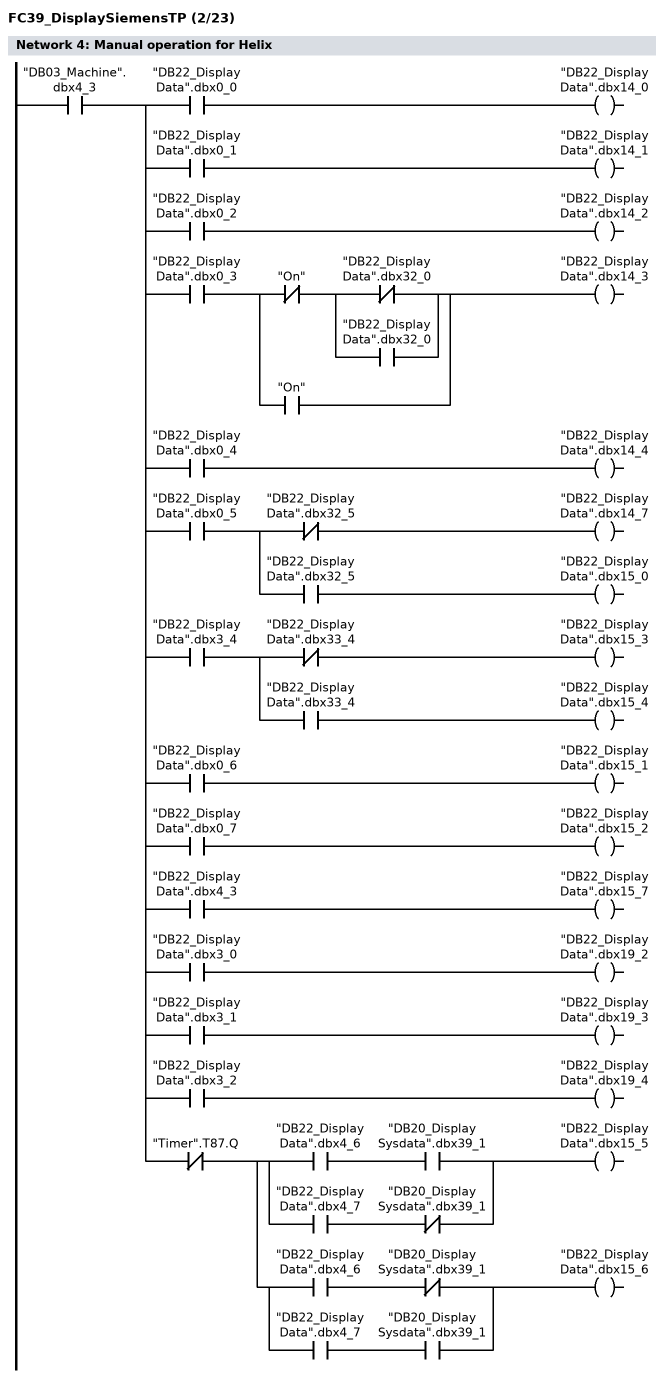
   RUNG wire#powerrail
      Contact( "DB03_Machine".dbx4_3 )
      wire#w1
      Contact( "DB22_DisplayData".dbx0_0 )
      Coil( "DB22_DisplayData".dbx14_0 )
   END_RUNG
   RUNG wire#w1
      Contact( "DB22_DisplayData".dbx0_1 )
      Coil( "DB22_DisplayData".dbx14_1 )
   END_RUNG
   RUNG wire#w1
      Contact( "DB22_DisplayData".dbx0_2 )
      Coil( "DB22_DisplayData".dbx14_2 )
   END_RUNG
   RUNG wire#w1
      Contact( "DB22_DisplayData".dbx0_3 )
      wire#w2
      I_Contact( "On" )
      wire#w3
      I_Contact( "DB22_DisplayData".dbx32_0 )
      wire#w4
      Coil( "DB22_DisplayData".dbx14_3 )
   END_RUNG
   RUNG wire#w3
      Contact( "DB22_DisplayData".dbx32_0 )
   END_RUNG wire#w4
   RUNG wire#w2
      Contact( "On" )
   END_RUNG wire#w4
   RUNG wire#w1
      Contact( "DB22_DisplayData".dbx0_4 )
      Coil( "DB22_DisplayData".dbx14_4 )
   END_RUNG
   RUNG wire#w1
      Contact( "DB22_DisplayData".dbx0_5 )
      wire#w5
      I_Contact( "DB22_DisplayData".dbx32_5 )
      Coil( "DB22_DisplayData".dbx14_7 )
   END_RUNG
   RUNG wire#w5
      Contact( "DB22_DisplayData".dbx32_5 )
      Coil( "DB22_DisplayData".dbx15_0 )
   END_RUNG
   RUNG wire#w1
      Contact( "DB22_DisplayData".dbx3_4 )
      wire#w6
      I_Contact( "DB22_DisplayData".dbx33_4 )
      Coil( "DB22_DisplayData".dbx15_3 )
   END_RUNG
   RUNG wire#w6
      Contact( "DB22_DisplayData".dbx33_4 )
      Coil( "DB22_DisplayData".dbx15_4 )
   END_RUNG
   RUNG wire#w1
      Contact( "DB22_DisplayData".dbx0_6 )
      Coil( "DB22_DisplayData".dbx15_1 )
   END_RUNG
   RUNG wire#w1
      Contact( "DB22_DisplayData".dbx0_7 )
      Coil( "DB22_DisplayData".dbx15_2 )
   END_RUNG
   RUNG wire#w1
      Contact( "DB22_DisplayData".dbx4_3 )
      Coil( "DB22_DisplayData".dbx15_7 )
   END_RUNG
   RUNG wire#w1
      Contact( "DB22_DisplayData".dbx3_0 )
      Coil( "DB22_DisplayData".dbx19_2 )
   END_RUNG
   RUNG wire#w1
      Contact( "DB22_DisplayData".dbx3_1 )
      Coil( "DB22_DisplayData".dbx19_3 )
   END_RUNG
   RUNG wire#w1
      Contact( "DB22_DisplayData".dbx3_2 )
      Coil( "DB22_DisplayData".dbx19_4 )
   END_RUNG
   RUNG wire#w1
      I_Contact( "Timer".T87.Q )
      wire#w7
      Contact( "DB22_DisplayData".dbx4_6 )
      Contact( "DB20_DisplaySysdata".dbx39_1 )
      wire#w8
      Coil( "DB22_DisplayData".dbx15_5 )
   END_RUNG
   RUNG wire#w7
      Contact( "DB22_DisplayData".dbx4_7 )
      I_Contact( "DB20_DisplaySysdata".dbx39_1 )
   END_RUNG wire#w8
   RUNG wire#w7
      Contact( "DB22_DisplayData".dbx4_6 )
      I_Contact( "DB20_DisplaySysdata".dbx39_1 )
      wire#w9
      Coil( "DB22_DisplayData".dbx15_6 )
   END_RUNG
   RUNG wire#w7
      Contact( "DB22_DisplayData".dbx4_7 )
      Contact( "DB20_DisplaySysdata".dbx39_1 )
   END_RUNG wire#w9
   // the same network as SCL:
   "DB22_DisplayData".dbx14_0 := "DB03_Machine".dbx4_3 AND "DB22_DisplayData".dbx0_0;
   "DB22_DisplayData".dbx14_1 := "DB03_Machine".dbx4_3 AND "DB22_DisplayData".dbx0_1;
   "DB22_DisplayData".dbx14_2 := "DB03_Machine".dbx4_3 AND "DB22_DisplayData".dbx0_2;
   "DB22_DisplayData".dbx14_3 := "DB03_Machine".dbx4_3 AND "DB22_DisplayData".dbx0_3 AND ((NOT "On" AND (NOT "DB22_DisplayData".dbx32_0 OR "DB22_DisplayData".dbx32_0)) OR "On");
   "DB22_DisplayData".dbx14_4 := "DB03_Machine".dbx4_3 AND "DB22_DisplayData".dbx0_4;
   #_w1 := "DB03_Machine".dbx4_3 AND "DB22_DisplayData".dbx0_5;
   "DB22_DisplayData".dbx14_7 := #_w1 AND NOT "DB22_DisplayData".dbx32_5;
   "DB22_DisplayData".dbx15_0 := #_w1 AND "DB22_DisplayData".dbx32_5;
   #_w2 := "DB03_Machine".dbx4_3 AND "DB22_DisplayData".dbx3_4;
   "DB22_DisplayData".dbx15_3 := #_w2 AND NOT "DB22_DisplayData".dbx33_4;
   "DB22_DisplayData".dbx15_4 := #_w2 AND "DB22_DisplayData".dbx33_4;
   "DB22_DisplayData".dbx15_1 := "DB03_Machine".dbx4_3 AND "DB22_DisplayData".dbx0_6;
   "DB22_DisplayData".dbx15_2 := "DB03_Machine".dbx4_3 AND "DB22_DisplayData".dbx0_7;
   "DB22_DisplayData".dbx15_7 := "DB03_Machine".dbx4_3 AND "DB22_DisplayData".dbx4_3;
   "DB22_DisplayData".dbx19_2 := "DB03_Machine".dbx4_3 AND "DB22_DisplayData".dbx3_0;
   "DB22_DisplayData".dbx19_3 := "DB03_Machine".dbx4_3 AND "DB22_DisplayData".dbx3_1;
   "DB22_DisplayData".dbx19_4 := "DB03_Machine".dbx4_3 AND "DB22_DisplayData".dbx3_2;
   #_w3 := "DB03_Machine".dbx4_3 AND NOT "Timer".T87.Q;
   "DB22_DisplayData".dbx15_5 := #_w3 AND (("DB22_DisplayData".dbx4_6 AND "DB20_DisplaySysdata".dbx39_1) OR ("DB22_DisplayData".dbx4_7 AND NOT "DB20_DisplaySysdata".dbx39_1));
   "DB22_DisplayData".dbx15_6 := #_w3 AND (("DB22_DisplayData".dbx4_6 AND NOT "DB20_DisplaySysdata".dbx39_1) OR ("DB22_DisplayData".dbx4_7 AND "DB20_DisplaySysdata".dbx39_1));
END_REGION

REGION Network 5: Manual(Toggle bit): Clamp upward/downward (Clamp)
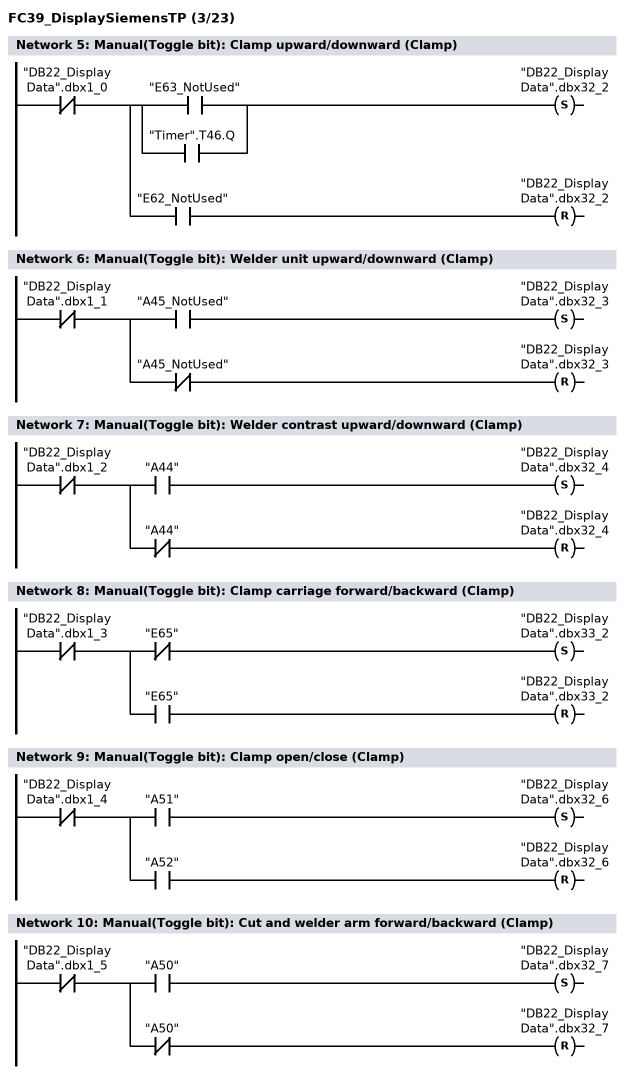
   RUNG wire#powerrail
      I_Contact( "DB22_DisplayData".dbx1_0 )
      wire#w1
      Contact( "E63_NotUsed" )
      wire#w2
      S_Coil( "DB22_DisplayData".dbx32_2 )
   END_RUNG
   RUNG wire#w1
      Contact( "Timer".T46.Q )
   END_RUNG wire#w2
   RUNG wire#w1
      Contact( "E62_NotUsed" )
      R_Coil( "DB22_DisplayData".dbx32_2 )
   END_RUNG
   // the same network as SCL:
   #_w1 := NOT "DB22_DisplayData".dbx1_0;
   IF #_w1 AND ("E63_NotUsed" OR "Timer".T46.Q) THEN "DB22_DisplayData".dbx32_2 := TRUE; END_IF;
   IF #_w1 AND "E62_NotUsed" THEN "DB22_DisplayData".dbx32_2 := FALSE; END_IF;
END_REGION

REGION Network 6: Manual(Toggle bit): Welder unit upward/downward (Clamp)
   RUNG wire#powerrail
      I_Contact( "DB22_DisplayData".dbx1_1 )
      wire#w1
      Contact( "A45_NotUsed" )
      S_Coil( "DB22_DisplayData".dbx32_3 )
   END_RUNG
   RUNG wire#w1
      I_Contact( "A45_NotUsed" )
      R_Coil( "DB22_DisplayData".dbx32_3 )
   END_RUNG
   // the same network as SCL:
   #_w1 := NOT "DB22_DisplayData".dbx1_1;
   IF #_w1 AND "A45_NotUsed" THEN "DB22_DisplayData".dbx32_3 := TRUE; END_IF;
   IF #_w1 AND NOT "A45_NotUsed" THEN "DB22_DisplayData".dbx32_3 := FALSE; END_IF;
END_REGION

REGION Network 7: Manual(Toggle bit): Welder contrast upward/downward (Clamp)
   RUNG wire#powerrail
      I_Contact( "DB22_DisplayData".dbx1_2 )
      wire#w1
      Contact( "A44" )
      S_Coil( "DB22_DisplayData".dbx32_4 )
   END_RUNG
   RUNG wire#w1
      I_Contact( "A44" )
      R_Coil( "DB22_DisplayData".dbx32_4 )
   END_RUNG
   // the same network as SCL:
   #_w1 := NOT "DB22_DisplayData".dbx1_2;
   IF #_w1 AND "A44" THEN "DB22_DisplayData".dbx32_4 := TRUE; END_IF;
   IF #_w1 AND NOT "A44" THEN "DB22_DisplayData".dbx32_4 := FALSE; END_IF;
END_REGION

REGION Network 8: Manual(Toggle bit): Clamp carriage forward/backward (Clamp)
   RUNG wire#powerrail
      I_Contact( "DB22_DisplayData".dbx1_3 )
      wire#w1
      I_Contact( "E65" )
      S_Coil( "DB22_DisplayData".dbx33_2 )
   END_RUNG
   RUNG wire#w1
      Contact( "E65" )
      R_Coil( "DB22_DisplayData".dbx33_2 )
   END_RUNG
   // the same network as SCL:
   #_w1 := NOT "DB22_DisplayData".dbx1_3;
   IF #_w1 AND NOT "E65" THEN "DB22_DisplayData".dbx33_2 := TRUE; END_IF;
   IF #_w1 AND "E65" THEN "DB22_DisplayData".dbx33_2 := FALSE; END_IF;
END_REGION

REGION Network 9: Manual(Toggle bit): Clamp open/close (Clamp)
   RUNG wire#powerrail
      I_Contact( "DB22_DisplayData".dbx1_4 )
      wire#w1
      Contact( "A51" )
      S_Coil( "DB22_DisplayData".dbx32_6 )
   END_RUNG
   RUNG wire#w1
      Contact( "A52" )
      R_Coil( "DB22_DisplayData".dbx32_6 )
   END_RUNG
   // the same network as SCL:
   #_w1 := NOT "DB22_DisplayData".dbx1_4;
   IF #_w1 AND "A51" THEN "DB22_DisplayData".dbx32_6 := TRUE; END_IF;
   IF #_w1 AND "A52" THEN "DB22_DisplayData".dbx32_6 := FALSE; END_IF;
END_REGION

REGION Network 10: Manual(Toggle bit): Cut and welder arm forward/backward (Clamp)
   RUNG wire#powerrail
      I_Contact( "DB22_DisplayData".dbx1_5 )
      wire#w1
      Contact( "A50" )
      S_Coil( "DB22_DisplayData".dbx32_7 )
   END_RUNG
   RUNG wire#w1
      I_Contact( "A50" )
      R_Coil( "DB22_DisplayData".dbx32_7 )
   END_RUNG
   // the same network as SCL:
   #_w1 := NOT "DB22_DisplayData".dbx1_5;
   IF #_w1 AND "A50" THEN "DB22_DisplayData".dbx32_7 := TRUE; END_IF;
   IF #_w1 AND NOT "A50" THEN "DB22_DisplayData".dbx32_7 := FALSE; END_IF;
END_REGION

REGION Network 11: Manual operation for clamp unit
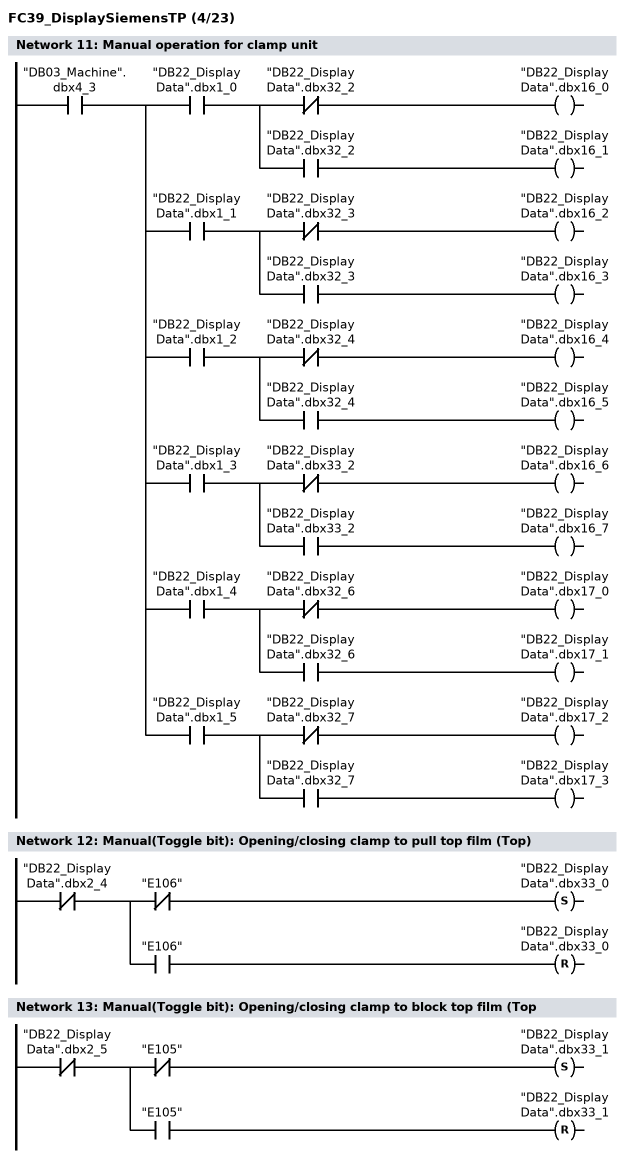
   RUNG wire#powerrail
      Contact( "DB03_Machine".dbx4_3 )
      wire#w1
      Contact( "DB22_DisplayData".dbx1_0 )
      wire#w2
      I_Contact( "DB22_DisplayData".dbx32_2 )
      Coil( "DB22_DisplayData".dbx16_0 )
   END_RUNG
   RUNG wire#w2
      Contact( "DB22_DisplayData".dbx32_2 )
      Coil( "DB22_DisplayData".dbx16_1 )
   END_RUNG
   RUNG wire#w1
      Contact( "DB22_DisplayData".dbx1_1 )
      wire#w3
      I_Contact( "DB22_DisplayData".dbx32_3 )
      Coil( "DB22_DisplayData".dbx16_2 )
   END_RUNG
   RUNG wire#w3
      Contact( "DB22_DisplayData".dbx32_3 )
      Coil( "DB22_DisplayData".dbx16_3 )
   END_RUNG
   RUNG wire#w1
      Contact( "DB22_DisplayData".dbx1_2 )
      wire#w4
      I_Contact( "DB22_DisplayData".dbx32_4 )
      Coil( "DB22_DisplayData".dbx16_4 )
   END_RUNG
   RUNG wire#w4
      Contact( "DB22_DisplayData".dbx32_4 )
      Coil( "DB22_DisplayData".dbx16_5 )
   END_RUNG
   RUNG wire#w1
      Contact( "DB22_DisplayData".dbx1_3 )
      wire#w5
      I_Contact( "DB22_DisplayData".dbx33_2 )
      Coil( "DB22_DisplayData".dbx16_6 )
   END_RUNG
   RUNG wire#w5
      Contact( "DB22_DisplayData".dbx33_2 )
      Coil( "DB22_DisplayData".dbx16_7 )
   END_RUNG
   RUNG wire#w1
      Contact( "DB22_DisplayData".dbx1_4 )
      wire#w6
      I_Contact( "DB22_DisplayData".dbx32_6 )
      Coil( "DB22_DisplayData".dbx17_0 )
   END_RUNG
   RUNG wire#w6
      Contact( "DB22_DisplayData".dbx32_6 )
      Coil( "DB22_DisplayData".dbx17_1 )
   END_RUNG
   RUNG wire#w1
      Contact( "DB22_DisplayData".dbx1_5 )
      wire#w7
      I_Contact( "DB22_DisplayData".dbx32_7 )
      Coil( "DB22_DisplayData".dbx17_2 )
   END_RUNG
   RUNG wire#w7
      Contact( "DB22_DisplayData".dbx32_7 )
      Coil( "DB22_DisplayData".dbx17_3 )
   END_RUNG
   // the same network as SCL:
   #_w1 := "DB03_Machine".dbx4_3 AND "DB22_DisplayData".dbx1_0;
   "DB22_DisplayData".dbx16_0 := #_w1 AND NOT "DB22_DisplayData".dbx32_2;
   "DB22_DisplayData".dbx16_1 := #_w1 AND "DB22_DisplayData".dbx32_2;
   #_w2 := "DB03_Machine".dbx4_3 AND "DB22_DisplayData".dbx1_1;
   "DB22_DisplayData".dbx16_2 := #_w2 AND NOT "DB22_DisplayData".dbx32_3;
   "DB22_DisplayData".dbx16_3 := #_w2 AND "DB22_DisplayData".dbx32_3;
   #_w3 := "DB03_Machine".dbx4_3 AND "DB22_DisplayData".dbx1_2;
   "DB22_DisplayData".dbx16_4 := #_w3 AND NOT "DB22_DisplayData".dbx32_4;
   "DB22_DisplayData".dbx16_5 := #_w3 AND "DB22_DisplayData".dbx32_4;
   #_w4 := "DB03_Machine".dbx4_3 AND "DB22_DisplayData".dbx1_3;
   "DB22_DisplayData".dbx16_6 := #_w4 AND NOT "DB22_DisplayData".dbx33_2;
   "DB22_DisplayData".dbx16_7 := #_w4 AND "DB22_DisplayData".dbx33_2;
   #_w5 := "DB03_Machine".dbx4_3 AND "DB22_DisplayData".dbx1_4;
   "DB22_DisplayData".dbx17_0 := #_w5 AND NOT "DB22_DisplayData".dbx32_6;
   "DB22_DisplayData".dbx17_1 := #_w5 AND "DB22_DisplayData".dbx32_6;
   #_w6 := "DB03_Machine".dbx4_3 AND "DB22_DisplayData".dbx1_5;
   "DB22_DisplayData".dbx17_2 := #_w6 AND NOT "DB22_DisplayData".dbx32_7;
   "DB22_DisplayData".dbx17_3 := #_w6 AND "DB22_DisplayData".dbx32_7;
END_REGION

REGION Network 12: Manual(Toggle bit): Opening/closing clamp to pull top film (Top)
   RUNG wire#powerrail
      I_Contact( "DB22_DisplayData".dbx2_4 )
      wire#w1
      I_Contact( "E106" )
      S_Coil( "DB22_DisplayData".dbx33_0 )
   END_RUNG
   RUNG wire#w1
      Contact( "E106" )
      R_Coil( "DB22_DisplayData".dbx33_0 )
   END_RUNG
   // the same network as SCL:
   #_w1 := NOT "DB22_DisplayData".dbx2_4;
   IF #_w1 AND NOT "E106" THEN "DB22_DisplayData".dbx33_0 := TRUE; END_IF;
   IF #_w1 AND "E106" THEN "DB22_DisplayData".dbx33_0 := FALSE; END_IF;
END_REGION

REGION Network 13: Manual(Toggle bit): Opening/closing clamp to block top film (Top
   RUNG wire#powerrail
      I_Contact( "DB22_DisplayData".dbx2_5 )
      wire#w1
      I_Contact( "E105" )
      S_Coil( "DB22_DisplayData".dbx33_1 )
   END_RUNG
   RUNG wire#w1
      Contact( "E105" )
      R_Coil( "DB22_DisplayData".dbx33_1 )
   END_RUNG
   // the same network as SCL:
   #_w1 := NOT "DB22_DisplayData".dbx2_5;
   IF #_w1 AND NOT "E105" THEN "DB22_DisplayData".dbx33_1 := TRUE; END_IF;
   IF #_w1 AND "E105" THEN "DB22_DisplayData".dbx33_1 := FALSE; END_IF;
END_REGION

REGION Network 14: Maual operation for top unit
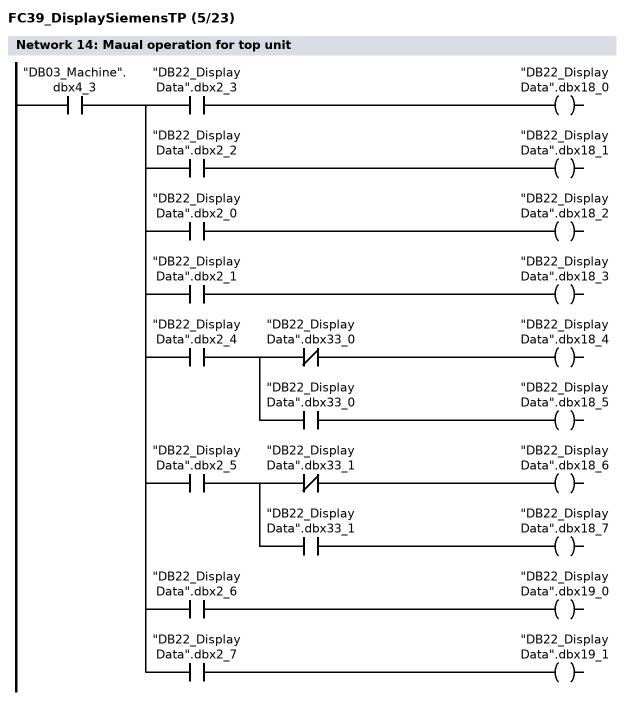
   RUNG wire#powerrail
      Contact( "DB03_Machine".dbx4_3 )
      wire#w1
      Contact( "DB22_DisplayData".dbx2_3 )
      Coil( "DB22_DisplayData".dbx18_0 )
   END_RUNG
   RUNG wire#w1
      Contact( "DB22_DisplayData".dbx2_2 )
      Coil( "DB22_DisplayData".dbx18_1 )
   END_RUNG
   RUNG wire#w1
      Contact( "DB22_DisplayData".dbx2_0 )
      Coil( "DB22_DisplayData".dbx18_2 )
   END_RUNG
   RUNG wire#w1
      Contact( "DB22_DisplayData".dbx2_1 )
      Coil( "DB22_DisplayData".dbx18_3 )
   END_RUNG
   RUNG wire#w1
      Contact( "DB22_DisplayData".dbx2_4 )
      wire#w2
      I_Contact( "DB22_DisplayData".dbx33_0 )
      Coil( "DB22_DisplayData".dbx18_4 )
   END_RUNG
   RUNG wire#w2
      Contact( "DB22_DisplayData".dbx33_0 )
      Coil( "DB22_DisplayData".dbx18_5 )
   END_RUNG
   RUNG wire#w1
      Contact( "DB22_DisplayData".dbx2_5 )
      wire#w3
      I_Contact( "DB22_DisplayData".dbx33_1 )
      Coil( "DB22_DisplayData".dbx18_6 )
   END_RUNG
   RUNG wire#w3
      Contact( "DB22_DisplayData".dbx33_1 )
      Coil( "DB22_DisplayData".dbx18_7 )
   END_RUNG
   RUNG wire#w1
      Contact( "DB22_DisplayData".dbx2_6 )
      Coil( "DB22_DisplayData".dbx19_0 )
   END_RUNG
   RUNG wire#w1
      Contact( "DB22_DisplayData".dbx2_7 )
      Coil( "DB22_DisplayData".dbx19_1 )
   END_RUNG
   // the same network as SCL:
   "DB22_DisplayData".dbx18_0 := "DB03_Machine".dbx4_3 AND "DB22_DisplayData".dbx2_3;
   "DB22_DisplayData".dbx18_1 := "DB03_Machine".dbx4_3 AND "DB22_DisplayData".dbx2_2;
   "DB22_DisplayData".dbx18_2 := "DB03_Machine".dbx4_3 AND "DB22_DisplayData".dbx2_0;
   "DB22_DisplayData".dbx18_3 := "DB03_Machine".dbx4_3 AND "DB22_DisplayData".dbx2_1;
   #_w1 := "DB03_Machine".dbx4_3 AND "DB22_DisplayData".dbx2_4;
   "DB22_DisplayData".dbx18_4 := #_w1 AND NOT "DB22_DisplayData".dbx33_0;
   "DB22_DisplayData".dbx18_5 := #_w1 AND "DB22_DisplayData".dbx33_0;
   #_w2 := "DB03_Machine".dbx4_3 AND "DB22_DisplayData".dbx2_5;
   "DB22_DisplayData".dbx18_6 := #_w2 AND NOT "DB22_DisplayData".dbx33_1;
   "DB22_DisplayData".dbx18_7 := #_w2 AND "DB22_DisplayData".dbx33_1;
   "DB22_DisplayData".dbx19_0 := "DB03_Machine".dbx4_3 AND "DB22_DisplayData".dbx2_6;
   "DB22_DisplayData".dbx19_1 := "DB03_Machine".dbx4_3 AND "DB22_DisplayData".dbx2_7;
END_REGION

REGION Network 15: Diagnostic signal conveyor
